LIN {X 0,Y 720.147,Z 331.518,A -85,B 0,C 180,E1 -1471.751,E2 -1471.751} C_VEL
LIN {X 0,Y 720.168,Z 331.521,A -85,B 0,C 180,E1 -1474.312,E2 -1474.312} C_VEL
LIN {X 0,Y 720.178,Z 331.516,A -85,B 0,C 180,E1 -1477.424,E2 -1477.424} C_VEL
LIN {X 0,Y 720.147,Z 331.52,A -85,B 0,C 180,E1 -1480.005,E2 -1480.005} C_VEL
LIN {X 0,Y 720.202,Z 331.519,A -85,B 0,C 180,E1 -1482.741,E2 -1482.741} C_VEL
LIN {X 0,Y 720.163,Z 331.518,A -85,B 0,C 180,E1 -1485.703,E2 -1485.703} C_VEL
LIN {X 0,Y 720.148,Z 331.521,A -85,B 0,C 180,E1 -1488.211,E2 -1488.211} C_VEL
LIN {X 0,Y 720.224,Z 331.522,A -85,B 0,C 180,E1 -1491.031,E2 -1491.031} C_VEL
LIN {X 0,Y 720.178,Z 331.658,A -85,B 0,C 180,E1 -1491.842,E2 -1491.842} C_VEL
LIN {X 0,Y 724.726,Z 343.938,A -85,B 0,C 180,E1 -1493.02,E2 -1493.02} C_VEL
LIN {X 0,Y 724.3,Z 377.38,A -85,B 0,C 180,E1 -1495.364,E2 -1495.364} C_VEL
LIN {X 0,Y 726.479,Z 386.984,A -85,B 0,C 180,E1 -1495.595,E2 -1495.595} C_VEL
LIN {X 0,Y 725.423,Z 646.459,A -85,B 0,C 180,E1 -1498.538,E2 -1498.538} C_VEL
LIN {X 0,Y 724.936,Z 767.067,A -85,B 0,C 180,E1 -1499.901,E2 -1499.901} C_VEL
LIN {X 0,Y 724.615,Z 792.768,A -85,B 0,C 180,E1 -1500.336,E2 -1500.336} C_VEL
LIN {X 0,Y 724.343,Z 814.337,A -85,B 0,C 180,E1 -1500.838,E2 -1500.838} C_VEL
LIN {X 0,Y 723.978,Z 838.571,A -85,B 0,C 180,E1 -1501.544,E2 -1501.544} C_VEL
LIN {X 0,Y 723.547,Z 860.481,A -85,B 0,C 180,E1 -1502.333,E2 -1502.333} C_VEL
LIN {X 0,Y 723.146,Z 883.179,A -85,B 0,C 180,E1 -1503.296,E2 -1503.296} C_VEL
LIN {X 0,Y 722.632,Z 904.752,A -85,B 0,C 180,E1 -1504.38,E2 -1504.38} C_VEL
LIN {X 0,Y 722.216,Z 925.848,A -85,B 0,C 180,E1 -1505.596,E2 -1505.596} C_VEL
LIN {X 0,Y 721.746,Z 945.564,A -85,B 0,C 180,E1 -1506.911,E2 -1506.911} C_VEL
LIN {X 0,Y 721.365,Z 964.778,A -85,B 0,C 180,E1 -1508.364,E2 -1508.364} C_VEL
LIN {X 0,Y 721.012,Z 981.391,A -85,B 0,C 180,E1 -1509.799,E2 -1509.799} C_VEL
LIN {X 0,Y 720.713,Z 998.517,A -85,B 0,C 180,E1 -1511.476,E2 -1511.476} C_VEL
LIN {X 0,Y 720.475,Z 1012.01,A -85,B 0,C 180,E1 -1512.982,E2 -1512.982} C_VEL
LIN {X 0,Y 720.287,Z 1026.218,A -85,B 0,C 180,E1 -1514.789,E2 -1514.789} C_VEL
LIN {X 0,Y 720.15,Z 1037.315,A -85,B 0,C 180,E1 -1516.429,E2 -1516.429} C_VEL
LIN {X 0,Y 720.044,Z 1047.962,A -85,B 0,C 180,E1 -1518.238,E2 -1518.238} C_VEL
LIN {X 0,Y 719.96,Z 1056.892,A -85,B 0,C 180,E1 -1520.083,E2 -1520.083} C_VEL
LIN {X 0,Y 719.941,Z 1063.423,A -85,B 0,C 180,E1 -1521.695,E2 -1521.695} C_VEL
LIN {X 0,Y 719.913,Z 1069.864,A -85,B 0,C 180,E1 -1523.701,E2 -1523.701} C_VEL
LIN {X 0,Y 719.916,Z 1073.813,A -85,B 0,C 180,E1 -1525.379,E2 -1525.379} C_VEL
LIN {X 0,Y 719.907,Z 1076.797,A -85,B 0,C 180,E1 -1527.214,E2 -1527.214} C_VEL
LIN {X 0,Y 719.9,Z 1078.284,A -85,B 0,C 180,E1 -1529.204,E2 -1529.204} C_VEL
LIN {X 0,Y 719.906,Z 1078.262,A -85,B 0,C 180,E1 -1530.875,E2 -1530.875} C_VEL
LIN {X 0,Y 719.913,Z 1076.572,A -85,B 0,C 180,E1 -1532.946,E2 -1532.946} C_VEL
LIN {X 0,Y 719.919,Z 1073.654,A -85,B 0,C 180,E1 -1534.7,E2 -1534.7} C_VEL
LIN {X 0,Y 719.908,Z 1069.015,A -85,B 0,C 180,E1 -1536.62,E2 -1536.62} C_VEL
LIN {X 0,Y 719.933,Z 1062.815,A -85,B 0,C 180,E1 -1538.466,E2 -1538.466} C_VEL
LIN {X 0,Y 719.974,Z 1056.182,A -85,B 0,C 180,E1 -1540.078,E2 -1540.078} C_VEL
LIN {X 0,Y 720.049,Z 1046.492,A -85,B 0,C 180,E1 -1542.023,E2 -1542.023} C_VEL
LIN {X 0,Y 720.154,Z 1036.797,A -85,B 0,C 180,E1 -1543.653,E2 -1543.653} C_VEL
LIN {X 0,Y 720.323,Z 1024.443,A -85,B 0,C 180,E1 -1545.457,E2 -1545.457} C_VEL
LIN {X 0,Y 720.483,Z 1011.22,A -85,B 0,C 180,E1 -1547.11,E2 -1547.11} C_VEL
LIN {X 0,Y 720.769,Z 996.177,A -85,B 0,C 180,E1 -1548.774,E2 -1548.774} C_VEL
LIN {X 0,Y 721.055,Z 979.533,A -85,B 0,C 180,E1 -1550.369,E2 -1550.369} C_VEL
LIN {X 0,Y 721.431,Z 961.605,A -85,B 0,C 180,E1 -1551.89,E2 -1551.89} C_VEL
LIN {X 0,Y 721.806,Z 943.237,A -85,B 0,C 180,E1 -1553.253,E2 -1553.253} C_VEL
LIN {X 0,Y 722.274,Z 921.436,A -85,B 0,C 180,E1 -1554.67,E2 -1554.67} C_VEL
LIN {X 0,Y 722.724,Z 901.528,A -85,B 0,C 180,E1 -1555.792,E2 -1555.792} C_VEL
LIN {X 0,Y 723.207,Z 878.257,A -85,B 0,C 180,E1 -1556.923,E2 -1556.923} C_VEL
LIN {X 0,Y 723.622,Z 857.111,A -85,B 0,C 180,E1 -1557.798,E2 -1557.798} C_VEL
LIN {X 0,Y 724.075,Z 832.965,A -85,B 0,C 180,E1 -1558.632,E2 -1558.632} C_VEL
LIN {X 0,Y 724.365,Z 811.104,A -85,B 0,C 180,E1 -1559.246,E2 -1559.246} C_VEL
LIN {X 0,Y 724.75,Z 786.45,A -85,B 0,C 180,E1 -1559.787,E2 -1559.787} C_VEL
LIN {X 0,Y 724.95,Z 763.827,A -85,B 0,C 180,E1 -1560.142,E2 -1560.142} C_VEL
LIN {X 0,Y 725.947,Z 508.76,A -85,B 0,C 180,E1 -1563.015,E2 -1563.015} C_VEL
LIN {X 0,Y 726.325,Z 385.42,A -85,B 0,C 180,E1 -1564.431,E2 -1564.431} C_VEL
LIN {X 0,Y 724.228,Z 376.685,A -85,B 0,C 180,E1 -1564.668,E2 -1564.668} C_VEL
LIN {X 0,Y 724.705,Z 343.756,A -85,B 0,C 180,E1 -1566.995,E2 -1566.995} C_VEL
LIN {X 0,Y 720.163,Z 331.523,A -85,B 0,C 180,E1 -1568.182,E2 -1568.182} C_VEL
LIN {X 0,Y 720.198,Z 331.524,A -85,B 0,C 180,E1 -1571.193,E2 -1571.193} C_VEL
LIN {X 0,Y 720.148,Z 331.521,A -85,B 0,C 180,E1 -1573.895,E2 -1573.895} C_VEL
LIN {X 0,Y 720.193,Z 331.517,A -85,B 0,C 180,E1 -1576.588,E2 -1576.588} C_VEL
LIN {X 0,Y 720.167,Z 331.519,A -85,B 0,C 180,E1 -1579.579,E2 -1579.579} C_VEL
LIN {X 0,Y 720.149,Z 331.518,A -85,B 0,C 180,E1 -1582.143,E2 -1582.143} C_VEL
LIN {X 0,Y 720.216,Z 331.516,A -85,B 0,C 180,E1 -1584.917,E2 -1584.917} C_VEL
LIN {X 0,Y 720.155,Z 331.519,A -85,B 0,C 180,E1 -1587.881,E2 -1587.881} C_VEL
LIN {X 0,Y 720.157,Z 331.517,A -85,B 0,C 180,E1 -1590.469,E2 -1590.469} C_VEL
LIN {X 0,Y 720.218,Z 331.517,A -85,B 0,C 180,E1 -1593.39,E2 -1593.39} C_VEL
LIN {X 0,Y 720.149,Z 331.515,A -85,B 0,C 180,E1 -1596.204,E2 -1596.204} C_VEL
LIN {X 0,Y 720.169,Z 331.516,A -85,B 0,C 180,E1 -1598.754,E2 -1598.754} C_VEL
LIN {X 0,Y 720.188,Z 331.521,A -85,B 0,C 180,E1 -1601.797,E2 -1601.797} C_VEL
LIN {X 0,Y 720.148,Z 331.517,A -85,B 0,C 180,E1 -1604.456,E2 -1604.456} C_VEL
LIN {X 0,Y 720.202,Z 331.513,A -85,B 0,C 180,E1 -1607.165,E2 -1607.165} C_VEL
LIN {X 0,Y 720.164,Z 331.515,A -85,B 0,C 180,E1 -1610.167,E2 -1610.167} C_VEL
LIN {X 0,Y 720.152,Z 331.517,A -85,B 0,C 180,E1 -1612.741,E2 -1612.741} C_VEL
LIN {X 0,Y 720.222,Z 331.515,A -85,B 0,C 180,E1 -1615.621,E2 -1615.621} C_VEL
LIN {X 0,Y 720.153,Z 331.519,A -85,B 0,C 180,E1 -1618.488,E2 -1618.488} C_VEL
LIN {X 0,Y 720.161,Z 331.511,A -85,B 0,C 180,E1 -1621.034,E2 -1621.034} C_VEL
LIN {X 0,Y 720.216,Z 331.521,A -85,B 0,C 180,E1 -1623.98,E2 -1623.98} C_VEL
LIN {X 0,Y 720.152,Z 331.517,A -85,B 0,C 180,E1 -1626.698,E2 -1626.698} C_VEL
LIN {X 0,Y 720.17,Z 331.516,A -85,B 0,C 180,E1 -1629.268,E2 -1629.268} C_VEL
LIN {X 0,Y 720.186,Z 331.521,A -85,B 0,C 180,E1 -1632.346,E2 -1632.346} C_VEL
LIN {X 0,Y 720.15,Z 331.516,A -85,B 0,C 180,E1 -1634.966,E2 -1634.966} C_VEL
LIN {X 0,Y 720.206,Z 331.518,A -85,B 0,C 180,E1 -1636.264,E2 -1636.264} C_VEL
LIN {X 0,Y 719.167,Z 331.649,A -85,B 0,C 180,E1 -1636.877,E2 -1636.877} C_VEL
LIN {X 0,Y 712.739,Z 332.448,A -85,B 0,C 180,E1 -1638.593,E2 -1638.593} C_VEL
LIN {X 0,Y 712.213,Z 332.507,A -85,B 0,C 180,E1 -1639.04,E2 -1639.04} C_VEL
LIN {X 0,Y 712.266,Z 332.499,A -85,B 0,C 180,E1 -1641.753,E2 -1641.753} C_VEL
LIN {X 0,Y 712.229,Z 332.504,A -85,B 0,C 180,E1 -1644.731,E2 -1644.731} C_VEL
LIN {X 0,Y 712.217,Z 332.506,A -85,B 0,C 180,E1 -1647.328,E2 -1647.328} C_VEL
LIN {X 0,Y 712.282,Z 332.501,A -85,B 0,C 180,E1 -1650.169,E2 -1650.169} C_VEL
LIN {X 0,Y 712.217,Z 332.505,A -85,B 0,C 180,E1 -1653.056,E2 -1653.056} C_VEL
LIN {X 0,Y 712.227,Z 332.505,A -85,B 0,C 180,E1 -1655.635,E2 -1655.635} C_VEL
LIN {X 0,Y 712.269,Z 332.51,A -85,B 0,C 180,E1 -1658.66,E2 -1658.66} C_VEL
LIN {X 0,Y 712.215,Z 332.509,A -85,B 0,C 180,E1 -1661.395,E2 -1661.395} C_VEL
LIN {X 0,Y 712.27,Z 332.495,A -85,B 0,C 180,E1 -1664.164,E2 -1664.164} C_VEL
LIN {X 0,Y 712.23,Z 332.509,A -85,B 0,C 180,E1 -1667.124,E2 -1667.124} C_VEL
LIN {X 0,Y 712.222,Z 332.508,A -85,B 0,C 180,E1 -1669.775,E2 -1669.775} C_VEL
LIN {X 0,Y 712.284,Z 332.51,A -85,B 0,C 180,E1 -1672.745,E2 -1672.745} C_VEL
LIN {X 0,Y 712.233,Z 332.633,A -85,B 0,C 180,E1 -1675.569,E2 -1675.569} C_VEL
LIN {X 0,Y 716.874,Z 346.258,A -85,B 0,C 180,E1 -1676.903,E2 -1676.903} C_VEL
LIN {X 0,Y 717.012,Z 348.148,A -85,B 0,C 180,E1 -1677.015,E2 -1677.015} C_VEL
LIN {X 0,Y 719.82,Z 359.326,A -85,B 0,C 180,E1 -1677.304,E2 -1677.304} C_VEL
LIN {X 0,Y 718.694,Z 595.051,A -85,B 0,C 180,E1 -1680.007,E2 -1680.007} C_VEL
LIN {X 0,Y 718.005,Z 736.964,A -85,B 0,C 180,E1 -1681.623,E2 -1681.623} C_VEL
LIN {X 0,Y 717.641,Z 762.526,A -85,B 0,C 180,E1 -1682.058,E2 -1682.058} C_VEL
LIN {X 0,Y 717.294,Z 784.203,A -85,B 0,C 180,E1 -1682.564,E2 -1682.564} C_VEL
LIN {X 0,Y 716.87,Z 808.198,A -85,B 0,C 180,E1 -1683.268,E2 -1683.268} C_VEL
LIN {X 0,Y 716.361,Z 829.733,A -85,B 0,C 180,E1 -1684.046,E2 -1684.046} C_VEL
LIN {X 0,Y 715.863,Z 852.405,A -85,B 0,C 180,E1 -1685.011,E2 -1685.011} C_VEL
LIN {X 0,Y 715.255,Z 874.42,A -85,B 0,C 180,E1 -1686.123,E2 -1686.123} C_VEL
LIN {X 0,Y 714.733,Z 895.263,A -85,B 0,C 180,E1 -1687.33,E2 -1687.33} C_VEL
LIN {X 0,Y 714.192,Z 914.96,A -85,B 0,C 180,E1 -1688.653,E2 -1688.653} C_VEL
LIN {X 0,Y 713.716,Z 933.972,A -85,B 0,C 180,E1 -1690.097,E2 -1690.097} C_VEL
LIN {X 0,Y 713.27,Z 951.38,A -85,B 0,C 180,E1 -1691.614,E2 -1691.614} C_VEL
LIN {X 0,Y 712.899,Z 968.676,A -85,B 0,C 180,E1 -1693.327,E2 -1693.327} C_VEL
LIN {X 0,Y 712.588,Z 983.029,A -85,B 0,C 180,E1 -1694.954,E2 -1694.954} C_VEL
LIN {X 0,Y 712.339,Z 997.581,A -85,B 0,C 180,E1 -1696.856,E2 -1696.856} C_VEL
LIN {X 0,Y 712.188,Z 1008.453,A -85,B 0,C 180,E1 -1698.5,E2 -1698.5} C_VEL
LIN {X 0,Y 712.068,Z 1019.527,A -85,B 0,C 180,E1 -1700.462,E2 -1700.462} C_VEL
LIN {X 0,Y 711.974,Z 1027.563,A -85,B 0,C 180,E1 -1702.171,E2 -1702.171} C_VEL
LIN {X 0,Y 711.944,Z 1034.871,A -85,B 0,C 180,E1 -1704.035,E2 -1704.035} C_VEL
LIN {X 0,Y 711.926,Z 1040.624,A -85,B 0,C 180,E1 -1705.973,E2 -1705.973} C_VEL
LIN {X 0,Y 711.916,Z 1044.548,A -85,B 0,C 180,E1 -1707.746,E2 -1707.746} C_VEL
LIN {X 0,Y 711.919,Z 1047.404,A -85,B 0,C 180,E1 -1709.839,E2 -1709.839} C_VEL
LIN {X 0,Y 711.89,Z 1048.364,A -85,B 0,C 180,E1 -1711.529,E2 -1711.529} C_VEL
LIN {X 0,Y 711.901,Z 1048.059,A -85,B 0,C 180,E1 -1713.462,E2 -1713.462} C_VEL
LIN {X 0,Y 711.906,Z 1046.161,A -85,B 0,C 180,E1 -1715.319,E2 -1715.319} C_VEL
LIN {X 0,Y 711.921,Z 1043.062,A -85,B 0,C 180,E1 -1717.1,E2 -1717.1} C_VEL
LIN {X 0,Y 711.935,Z 1037.783,A -85,B 0,C 180,E1 -1719.132,E2 -1719.132} C_VEL
LIN {X 0,Y 711.938,Z 1032.221,A -85,B 0,C 180,E1 -1720.766,E2 -1720.766} C_VEL
LIN {X 0,Y 712.017,Z 1024.357,A -85,B 0,C 180,E1 -1722.655,E2 -1722.655} C_VEL
LIN {X 0,Y 712.112,Z 1014.976,A -85,B 0,C 180,E1 -1724.474,E2 -1724.474} C_VEL
LIN {X 0,Y 712.25,Z 1004.476,A -85,B 0,C 180,E1 -1726.222,E2 -1726.222} C_VEL
LIN {X 0,Y 712.441,Z 991.458,A -85,B 0,C 180,E1 -1728.069,E2 -1728.069} C_VEL
LIN {X 0,Y 712.708,Z 978.141,A -85,B 0,C 180,E1 -1729.715,E2 -1729.715} C_VEL
LIN {X 0,Y 713.004,Z 962.68,A -85,B 0,C 180,E1 -1731.384,E2 -1731.384} C_VEL
LIN {X 0,Y 713.401,Z 946.869,A -85,B 0,C 180,E1 -1732.889,E2 -1732.889} C_VEL
LIN {X 0,Y 713.83,Z 928.46,A -85,B 0,C 180,E1 -1734.427,E2 -1734.427} C_VEL
LIN {X 0,Y 714.333,Z 910.388,A -85,B 0,C 180,E1 -1735.761,E2 -1735.761} C_VEL
LIN {X 0,Y 714.844,Z 889.874,A -85,B 0,C 180,E1 -1737.084,E2 -1737.084} C_VEL
LIN {X 0,Y 715.391,Z 870.255,A -85,B 0,C 180,E1 -1738.191,E2 -1738.191} C_VEL
LIN {X 0,Y 715.937,Z 847.27,A -85,B 0,C 180,E1 -1739.309,E2 -1739.309} C_VEL
LIN {X 0,Y 716.445,Z 826.736,A -85,B 0,C 180,E1 -1740.161,E2 -1740.161} C_VEL
LIN {X 0,Y 716.974,Z 802.732,A -85,B 0,C 180,E1 -1740.994,E2 -1740.994} C_VEL
LIN {X 0,Y 717.328,Z 781.027,A -85,B 0,C 180,E1 -1741.608,E2 -1741.608} C_VEL
LIN {X 0,Y 717.788,Z 756.2,A -85,B 0,C 180,E1 -1742.155,E2 -1742.155} C_VEL
LIN {X 0,Y 718.022,Z 733.611,A -85,B 0,C 180,E1 -1742.511,E2 -1742.511} C_VEL
LIN {X 0,Y 719.275,Z 474.158,A -85,B 0,C 180,E1 -1745.46,E2 -1745.46} C_VEL
LIN {X 0,Y 719.66,Z 357.915,A -85,B 0,C 180,E1 -1746.811,E2 -1746.811} C_VEL
LIN {X 0,Y 716.859,Z 347.284,A -85,B 0,C 180,E1 -1747.109,E2 -1747.109} C_VEL
LIN {X 0,Y 716.355,Z 344.494,A -85,B 0,C 180,E1 -1747.353,E2 -1747.353} C_VEL
LIN {X 0,Y 712.215,Z 332.516,A -85,B 0,C 180,E1 -1748.56,E2 -1748.56} C_VEL
LIN {X 0,Y 712.284,Z 332.508,A -85,B 0,C 180,E1 -1751.442,E2 -1751.442} C_VEL
LIN {X 0,Y 712.216,Z 332.507,A -85,B 0,C 180,E1 -1754.359,E2 -1754.359} C_VEL
LIN {X 0,Y 712.233,Z 332.509,A -85,B 0,C 180,E1 -1757.006,E2 -1757.006} C_VEL
LIN {X 0,Y 712.245,Z 332.502,A -85,B 0,C 180,E1 -1760.091,E2 -1760.091} C_VEL
LIN {X 0,Y 712.213,Z 332.508,A -85,B 0,C 180,E1 -1762.752,E2 -1762.752} C_VEL
LIN {X 0,Y 712.278,Z 332.503,A -85,B 0,C 180,E1 -1765.547,E2 -1765.547} C_VEL
LIN {X 0,Y 712.219,Z 332.503,A -85,B 0,C 180,E1 -1768.516,E2 -1768.516} C_VEL
LIN {X 0,Y 712.224,Z 332.509,A -85,B 0,C 180,E1 -1771.122,E2 -1771.122} C_VEL
LIN {X 0,Y 712.272,Z 332.501,A -85,B 0,C 180,E1 -1774.114,E2 -1774.114} C_VEL
LIN {X 0,Y 712.213,Z 332.507,A -85,B 0,C 180,E1 -1776.863,E2 -1776.863} C_VEL
LIN {X 0,Y 712.249,Z 332.508,A -85,B 0,C 180,E1 -1779.54,E2 -1779.54} C_VEL
LIN {X 0,Y 712.23,Z 332.503,A -85,B 0,C 180,E1 -1782.601,E2 -1782.601} C_VEL
LIN {X 0,Y 712.213,Z 332.508,A -85,B 0,C 180,E1 -1785.196,E2 -1785.196} C_VEL
LIN {X 0,Y 712.283,Z 332.507,A -85,B 0,C 180,E1 -1788.079,E2 -1788.079} C_VEL
LIN {X 0,Y 712.216,Z 332.505,A -85,B 0,C 180,E1 -1790.953,E2 -1790.953} C_VEL
LIN {X 0,Y 712.225,Z 332.509,A -85,B 0,C 180,E1 -1793.551,E2 -1793.551} C_VEL
LIN {X 0,Y 712.266,Z 332.504,A -85,B 0,C 180,E1 -1796.539,E2 -1796.539} C_VEL
LIN {X 0,Y 712.21,Z 332.504,A -85,B 0,C 180,E1 -1799.276,E2 -1799.276} C_VEL
LIN {X 0,Y 712.249,Z 332.511,A -85,B 0,C 180,E1 -1801.931,E2 -1801.931} C_VEL
LIN {X 0,Y 712.228,Z 332.505,A -85,B 0,C 180,E1 -1804.993,E2 -1804.993} C_VEL
LIN {X 0,Y 712.211,Z 332.504,A -85,B 0,C 180,E1 -1807.583,E2 -1807.583} C_VEL
LIN {X 0,Y 712.283,Z 332.504,A -85,B 0,C 180,E1 -1810.433,E2 -1810.433} C_VEL
LIN {X 0,Y 712.216,Z 332.506,A -85,B 0,C 180,E1 -1813.311,E2 -1813.311} C_VEL
LIN {X 0,Y 712.221,Z 332.505,A -85,B 0,C 180,E1 -1815.914,E2 -1815.914} C_VEL
LIN {X 0,Y 712.263,Z 332.499,A -85,B 0,C 180,E1 -1818.922,E2 -1818.922} C_VEL
LIN {X 0,Y 712.209,Z 332.507,A -85,B 0,C 180,E1 -1821.668,E2 -1821.668} C_VEL
LIN {X 0,Y 712.252,Z 332.507,A -85,B 0,C 180,E1 -1824.343,E2 -1824.343} C_VEL
LIN {X 0,Y 712.231,Z 332.503,A -85,B 0,C 180,E1 -1827.327,E2 -1827.327} C_VEL
LIN {X 0,Y 712.209,Z 332.508,A -85,B 0,C 180,E1 -1829.894,E2 -1829.894} C_VEL
LIN {X 0,Y 712.28,Z 332.51,A -85,B 0,C 180,E1 -1832.715,E2 -1832.715} C_VEL
LIN {X 0,Y 712.218,Z 332.507,A -85,B 0,C 180,E1 -1835.635,E2 -1835.635} C_VEL
LIN {X 0,Y 712.214,Z 332.509,A -85,B 0,C 180,E1 -1838.169,E2 -1838.169} C_VEL
LIN {X 0,Y 712.283,Z 332.506,A -85,B 0,C 180,E1 -1841.077,E2 -1841.077} C_VEL
LIN {X 0,Y 712.21,Z 332.508,A -85,B 0,C 180,E1 -1843.928,E2 -1843.928} C_VEL
LIN {X 0,Y 712.231,Z 332.512,A -85,B 0,C 180,E1 -1846.537,E2 -1846.537} C_VEL
LIN {X 0,Y 712.234,Z 332.511,A -85,B 0,C 180,E1 -1849.67,E2 -1849.67} C_VEL
LIN {X 0,Y 712.304,Z 332.749,A -85,B 0,C 180,E1 -1851.434,E2 -1851.434} C_VEL
LIN {X 0,Y 717.694,Z 347.211,A -85,B 0,C 180,E1 -1852.836,E2 -1852.836} C_VEL
LIN {X 0,Y 717.276,Z 377.475,A -85,B 0,C 180,E1 -1854.976,E2 -1854.976} C_VEL
LIN {X 0,Y 719.862,Z 388.77,A -85,B 0,C 180,E1 -1855.255,E2 -1855.255} C_VEL
LIN {X 0,Y 718.585,Z 648.445,A -85,B 0,C 180,E1 -1858.226,E2 -1858.226} C_VEL
LIN {X 0,Y 718.004,Z 767.174,A -85,B 0,C 180,E1 -1859.581,E2 -1859.581} C_VEL
LIN {X 0,Y 717.629,Z 792.895,A -85,B 0,C 180,E1 -1860.021,E2 -1860.021} C_VEL
LIN {X 0,Y 717.291,Z 814.459,A -85,B 0,C 180,E1 -1860.526,E2 -1860.526} C_VEL
LIN {X 0,Y 716.861,Z 838.568,A -85,B 0,C 180,E1 -1861.235,E2 -1861.235} C_VEL
LIN {X 0,Y 716.339,Z 860.486,A -85,B 0,C 180,E1 -1862.031,E2 -1862.031} C_VEL
LIN {X 0,Y 715.831,Z 883.582,A -85,B 0,C 180,E1 -1863.022,E2 -1863.022} C_VEL
LIN {X 0,Y 715.246,Z 904.756,A -85,B 0,C 180,E1 -1864.096,E2 -1864.096} C_VEL
LIN {X 0,Y 714.719,Z 925.755,A -85,B 0,C 180,E1 -1865.317,E2 -1865.317} C_VEL
LIN {X 0,Y 714.177,Z 945.152,A -85,B 0,C 180,E1 -1866.622,E2 -1866.622} C_VEL
LIN {X 0,Y 713.724,Z 963.809,A -85,B 0,C 180,E1 -1868.038,E2 -1868.038} C_VEL
LIN {X 0,Y 713.296,Z 980.462,A -85,B 0,C 180,E1 -1869.485,E2 -1869.485} C_VEL
LIN {X 0,Y 712.938,Z 996.965,A -85,B 0,C 180,E1 -1871.096,E2 -1871.096} C_VEL
LIN {X 0,Y 712.623,Z 1011.222,A -85,B 0,C 180,E1 -1872.695,E2 -1872.695} C_VEL
LIN {X 0,Y 712.408,Z 1025.06,A -85,B 0,C 180,E1 -1874.45,E2 -1874.45} C_VEL
LIN {X 0,Y 712.209,Z 1036.797,A -85,B 0,C 180,E1 -1876.192,E2 -1876.192} C_VEL
LIN {X 0,Y 712.082,Z 1046.948,A -85,B 0,C 180,E1 -1877.923,E2 -1877.923} C_VEL
LIN {X 0,Y 711.99,Z 1056.524,A -85,B 0,C 180,E1 -1879.886,E2 -1879.886} C_VEL
LIN {X 0,Y 711.94,Z 1063.12,A -85,B 0,C 180,E1 -1881.52,E2 -1881.52} C_VEL
LIN {X 0,Y 711.909,Z 1069.451,A -85,B 0,C 180,E1 -1883.468,E2 -1883.468} C_VEL
LIN {X 0,Y 711.918,Z 1073.814,A -85,B 0,C 180,E1 -1885.327,E2 -1885.327} C_VEL
LIN {X 0,Y 711.908,Z 1076.797,A -85,B 0,C 180,E1 -1887.182,E2 -1887.182} C_VEL
LIN {X 0,Y 711.901,Z 1078.284,A -85,B 0,C 180,E1 -1889.195,E2 -1889.195} C_VEL
LIN {X 0,Y 711.906,Z 1078.262,A -85,B 0,C 180,E1 -1890.885,E2 -1890.885} C_VEL
LIN {X 0,Y 711.914,Z 1076.572,A -85,B 0,C 180,E1 -1892.979,E2 -1892.979} C_VEL
LIN {X 0,Y 711.919,Z 1073.655,A -85,B 0,C 180,E1 -1894.753,E2 -1894.753} C_VEL
LIN {X 0,Y 711.914,Z 1069.015,A -85,B 0,C 180,E1 -1896.694,E2 -1896.694} C_VEL
LIN {X 0,Y 711.938,Z 1062.815,A -85,B 0,C 180,E1 -1898.562,E2 -1898.562} C_VEL
LIN {X 0,Y 712.001,Z 1056.182,A -85,B 0,C 180,E1 -1900.192,E2 -1900.192} C_VEL
LIN {X 0,Y 712.095,Z 1046.032,A -85,B 0,C 180,E1 -1902.241,E2 -1902.241} C_VEL
LIN {X 0,Y 712.214,Z 1036.279,A -85,B 0,C 180,E1 -1903.891,E2 -1903.891} C_VEL
LIN {X 0,Y 712.423,Z 1023.806,A -85,B 0,C 180,E1 -1905.716,E2 -1905.716} C_VEL
LIN {X 0,Y 712.64,Z 1010.515,A -85,B 0,C 180,E1 -1907.389,E2 -1907.389} C_VEL
LIN {X 0,Y 712.961,Z 995.334,A -85,B 0,C 180,E1 -1909.073,E2 -1909.073} C_VEL
LIN {X 0,Y 713.319,Z 979.534,A -85,B 0,C 180,E1 -1910.6,E2 -1910.6} C_VEL
LIN {X 0,Y 713.767,Z 961.606,A -85,B 0,C 180,E1 -1912.138,E2 -1912.138} C_VEL
LIN {X 0,Y 714.239,Z 943.237,A -85,B 0,C 180,E1 -1913.515,E2 -1913.515} C_VEL
LIN {X 0,Y 714.782,Z 922.166,A -85,B 0,C 180,E1 -1914.902,E2 -1914.902} C_VEL
LIN {X 0,Y 715.321,Z 902.334,A -85,B 0,C 180,E1 -1916.035,E2 -1916.035} C_VEL
LIN {X 0,Y 715.904,Z 879.254,A -85,B 0,C 180,E1 -1917.175,E2 -1917.175} C_VEL
LIN {X 0,Y 716.401,Z 858.239,A -85,B 0,C 180,E1 -1918.057,E2 -1918.057} C_VEL
LIN {X 0,Y 716.951,Z 834.438,A -85,B 0,C 180,E1 -1918.897,E2 -1918.897} C_VEL
LIN {X 0,Y 717.314,Z 811.86,A -85,B 0,C 180,E1 -1919.542,E2 -1919.542} C_VEL
LIN {X 0,Y 717.775,Z 787.537,A -85,B 0,C 180,E1 -1920.087,E2 -1920.087} C_VEL
LIN {X 0,Y 718.02,Z 764.114,A -85,B 0,C 180,E1 -1920.459,E2 -1920.459} C_VEL
LIN {X 0,Y 719.22,Z 511.246,A -85,B 0,C 180,E1 -1923.334,E2 -1923.334} C_VEL
LIN {X 0,Y 719.678,Z 387.124,A -85,B 0,C 180,E1 -1924.775,E2 -1924.775} C_VEL
LIN {X 0,Y 717.183,Z 376.685,A -85,B 0,C 180,E1 -1925.058,E2 -1925.058} C_VEL
LIN {X 0,Y 717.695,Z 347.209,A -85,B 0,C 180,E1 -1927.164,E2 -1927.164} C_VEL
LIN {X 0,Y 712.276,Z 332.509,A -85,B 0,C 180,E1 -1928.608,E2 -1928.608} C_VEL
LIN {X 0,Y 712.219,Z 332.513,A -85,B 0,C 180,E1 -1931.558,E2 -1931.558} C_VEL
LIN {X 0,Y 712.214,Z 332.51,A -85,B 0,C 180,E1 -1934.134,E2 -1934.134} C_VEL
LIN {X 0,Y 712.281,Z 332.51,A -85,B 0,C 180,E1 -1937.001,E2 -1937.001} C_VEL
LIN {X 0,Y 712.213,Z 332.507,A -85,B 0,C 180,E1 -1939.794,E2 -1939.794} C_VEL
LIN {X 0,Y 712.219,Z 332.506,A -85,B 0,C 180,E1 -1942.36,E2 -1942.36} C_VEL
LIN {X 0,Y 712.271,Z 332.507,A -85,B 0,C 180,E1 -1945.351,E2 -1945.351} C_VEL
LIN {X 0,Y 712.209,Z 332.507,A -85,B 0,C 180,E1 -1948.043,E2 -1948.043} C_VEL
LIN {X 0,Y 712.234,Z 332.505,A -85,B 0,C 180,E1 -1950.669,E2 -1950.669} C_VEL
LIN {X 0,Y 712.236,Z 332.51,A -85,B 0,C 180,E1 -1953.776,E2 -1953.776} C_VEL
LIN {X 0,Y 712.211,Z 332.503,A -85,B 0,C 180,E1 -1956.414,E2 -1956.414} C_VEL
LIN {X 0,Y 712.282,Z 332.504,A -85,B 0,C 180,E1 -1959.215,E2 -1959.215} C_VEL
LIN {X 0,Y 712.218,Z 332.508,A -85,B 0,C 180,E1 -1962.148,E2 -1962.148} C_VEL
LIN {X 0,Y 712.218,Z 332.504,A -85,B 0,C 180,E1 -1964.696,E2 -1964.696} C_VEL
LIN {X 0,Y 712.282,Z 332.508,A -85,B 0,C 180,E1 -1967.597,E2 -1967.597} C_VEL
LIN {X 0,Y 712.212,Z 332.503,A -85,B 0,C 180,E1 -1970.383,E2 -1970.383} C_VEL
LIN {X 0,Y 712.231,Z 332.505,A -85,B 0,C 180,E1 -1973,E2 -1973} C_VEL
LIN {X 0,Y 712.238,Z 332.508,A -85,B 0,C 180,E1 -1976.136,E2 -1976.136} C_VEL
LIN {X 0,Y 712.214,Z 332.506,A -85,B 0,C 180,E1 -1978.793,E2 -1978.793} C_VEL
LIN {X 0,Y 712.283,Z 332.498,A -85,B 0,C 180,E1 -1981.609,E2 -1981.609} C_VEL
LIN {X 0,Y 712.219,Z 332.506,A -85,B 0,C 180,E1 -1984.509,E2 -1984.509} C_VEL
LIN {X 0,Y 712.22,Z 332.503,A -85,B 0,C 180,E1 -1987.097,E2 -1987.097} C_VEL
LIN {X 0,Y 712.28,Z 332.507,A -85,B 0,C 180,E1 -1990.025,E2 -1990.025} C_VEL
LIN {X 0,Y 712.213,Z 332.507,A -85,B 0,C 180,E1 -1992.816,E2 -1992.816} C_VEL
LIN {X 0,Y 712.233,Z 332.503,A -85,B 0,C 180,E1 -1995.387,E2 -1995.387} C_VEL
LIN {X 0,Y 712.242,Z 332.51,A -85,B 0,C 180,E1 -1998.498,E2 -1998.498} C_VEL
LIN {X 0,Y 712.213,Z 332.507,A -85,B 0,C 180,E1 -1999.04,E2 -1999.04} C_VEL
LIN {X 0,Y 711.228,Z 332.632,A -85,B 0,C 180,E1 -1999.659,E2 -1999.659} C_VEL
LIN {X 0,Y 704.842,Z 333.422,A -85,B 0,C 180,E1 -2001.395,E2 -2001.395} C_VEL
LIN {X 0,Y 704.336,Z 333.488,A -85,B 0,C 180,E1 -2001.847,E2 -2001.847} C_VEL
LIN {X 0,Y 704.281,Z 333.492,A -85,B 0,C 180,E1 -2004.85,E2 -2004.85} C_VEL
LIN {X 0,Y 704.286,Z 333.495,A -85,B 0,C 180,E1 -2007.478,E2 -2007.478} C_VEL
LIN {X 0,Y 704.333,Z 333.498,A -85,B 0,C 180,E1 -2010.491,E2 -2010.491} C_VEL
LIN {X 0,Y 704.275,Z 333.492,A -85,B 0,C 180,E1 -2013.256,E2 -2013.256} C_VEL
LIN {X 0,Y 704.328,Z 333.493,A -85,B 0,C 180,E1 -2015.996,E2 -2015.996} C_VEL
LIN {X 0,Y 704.286,Z 333.497,A -85,B 0,C 180,E1 -2019.051,E2 -2019.051} C_VEL
LIN {X 0,Y 704.284,Z 333.497,A -85,B 0,C 180,E1 -2021.688,E2 -2021.688} C_VEL
LIN {X 0,Y 704.338,Z 333.483,A -85,B 0,C 180,E1 -2024.665,E2 -2024.665} C_VEL
LIN {X 0,Y 704.278,Z 333.495,A -85,B 0,C 180,E1 -2027.484,E2 -2027.484} C_VEL
LIN {X 0,Y 704.322,Z 333.495,A -85,B 0,C 180,E1 -2030.189,E2 -2030.189} C_VEL
LIN {X 0,Y 704.296,Z 333.504,A -85,B 0,C 180,E1 -2033.199,E2 -2033.199} C_VEL
LIN {X 0,Y 704.318,Z 333.634,A -85,B 0,C 180,E1 -2035.172,E2 -2035.172} C_VEL
LIN {X 0,Y 709.413,Z 347.994,A -85,B 0,C 180,E1 -2036.582,E2 -2036.582} C_VEL
LIN {X 0,Y 710.976,Z 352.032,A -85,B 0,C 180,E1 -2036.72,E2 -2036.72} C_VEL
LIN {X 0,Y 713.228,Z 361.214,A -85,B 0,C 180,E1 -2036.959,E2 -2036.959} C_VEL
LIN {X 0,Y 711.899,Z 596.712,A -85,B 0,C 180,E1 -2039.683,E2 -2039.683} C_VEL
LIN {X 0,Y 711.095,Z 737.104,A -85,B 0,C 180,E1 -2041.298,E2 -2041.298} C_VEL
LIN {X 0,Y 710.683,Z 762.688,A -85,B 0,C 180,E1 -2041.738,E2 -2041.738} C_VEL
LIN {X 0,Y 710.264,Z 784.444,A -85,B 0,C 180,E1 -2042.25,E2 -2042.25} C_VEL
LIN {X 0,Y 709.748,Z 808.927,A -85,B 0,C 180,E1 -2042.978,E2 -2042.978} C_VEL
LIN {X 0,Y 709.162,Z 830.486,A -85,B 0,C 180,E1 -2043.767,E2 -2043.767} C_VEL
LIN {X 0,Y 708.547,Z 853.569,A -85,B 0,C 180,E1 -2044.766,E2 -2044.766} C_VEL
LIN {X 0,Y 707.876,Z 874.78,A -85,B 0,C 180,E1 -2045.852,E2 -2045.852} C_VEL
LIN {X 0,Y 707.217,Z 896.311,A -85,B 0,C 180,E1 -2047.12,E2 -2047.12} C_VEL
LIN {X 0,Y 706.618,Z 915.313,A -85,B 0,C 180,E1 -2048.413,E2 -2048.413} C_VEL
LIN {X 0,Y 706.049,Z 934.283,A -85,B 0,C 180,E1 -2049.873,E2 -2049.873} C_VEL
LIN {X 0,Y 705.564,Z 950.732,A -85,B 0,C 180,E1 -2051.32,E2 -2051.32} C_VEL
LIN {X 0,Y 705.13,Z 967.025,A -85,B 0,C 180,E1 -2052.931,E2 -2052.931} C_VEL
LIN {X 0,Y 704.75,Z 981.839,A -85,B 0,C 180,E1 -2054.614,E2 -2054.614} C_VEL
LIN {X 0,Y 704.487,Z 995.453,A -85,B 0,C 180,E1 -2056.373,E2 -2056.373} C_VEL
LIN {X 0,Y 704.269,Z 1007.058,A -85,B 0,C 180,E1 -2058.12,E2 -2058.12} C_VEL
LIN {X 0,Y 704.119,Z 1017.561,A -85,B 0,C 180,E1 -2059.941,E2 -2059.941} C_VEL
LIN {X 0,Y 704.013,Z 1026.732,A -85,B 0,C 180,E1 -2061.864,E2 -2061.864} C_VEL
LIN {X 0,Y 703.947,Z 1033.449,A -85,B 0,C 180,E1 -2063.557,E2 -2063.557} C_VEL
LIN {X 0,Y 703.921,Z 1040.067,A -85,B 0,C 180,E1 -2065.682,E2 -2065.682} C_VEL
LIN {X 0,Y 703.915,Z 1043.96,A -85,B 0,C 180,E1 -2067.395,E2 -2067.395} C_VEL
LIN {X 0,Y 703.899,Z 1046.897,A -85,B 0,C 180,E1 -2069.267,E2 -2069.267} C_VEL
LIN {X 0,Y 703.9,Z 1048.281,A -85,B 0,C 180,E1 -2071.221,E2 -2071.221} C_VEL
LIN {X 0,Y 703.906,Z 1048.264,A -85,B 0,C 180,E1 -2072.931,E2 -2072.931} C_VEL
LIN {X 0,Y 703.911,Z 1046.58,A -85,B 0,C 180,E1 -2075.053,E2 -2075.053} C_VEL
LIN {X 0,Y 703.91,Z 1043.716,A -85,B 0,C 180,E1 -2076.821,E2 -2076.821} C_VEL
LIN {X 0,Y 703.925,Z 1039.223,A -85,B 0,C 180,E1 -2078.742,E2 -2078.742} C_VEL
LIN {X 0,Y 703.944,Z 1033.051,A -85,B 0,C 180,E1 -2080.641,E2 -2080.641} C_VEL
LIN {X 0,Y 704.021,Z 1026.412,A -85,B 0,C 180,E1 -2082.3,E2 -2082.3} C_VEL
LIN {X 0,Y 704.132,Z 1016.7,A -85,B 0,C 180,E1 -2084.305,E2 -2084.305} C_VEL
LIN {X 0,Y 704.274,Z 1006.757,A -85,B 0,C 180,E1 -2086.018,E2 -2086.018} C_VEL
LIN {X 0,Y 704.507,Z 994.482,A -85,B 0,C 180,E1 -2087.852,E2 -2087.852} C_VEL
LIN {X 0,Y 704.771,Z 981.118,A -85,B 0,C 180,E1 -2089.562,E2 -2089.562} C_VEL
LIN {X 0,Y 705.153,Z 965.849,A -85,B 0,C 180,E1 -2091.285,E2 -2091.285} C_VEL
LIN {X 0,Y 705.59,Z 949.887,A -85,B 0,C 180,E1 -2092.848,E2 -2092.848} C_VEL
LIN {X 0,Y 706.101,Z 932.311,A -85,B 0,C 180,E1 -2094.38,E2 -2094.38} C_VEL
LIN {X 0,Y 706.671,Z 913.726,A -85,B 0,C 180,E1 -2095.791,E2 -2095.791} C_VEL
LIN {X 0,Y 707.3,Z 893.136,A -85,B 0,C 180,E1 -2097.169,E2 -2097.169} C_VEL
LIN {X 0,Y 707.937,Z 873.068,A -85,B 0,C 180,E1 -2098.331,E2 -2098.331} C_VEL
LIN {X 0,Y 708.616,Z 850.437,A -85,B 0,C 180,E1 -2099.469,E2 -2099.469} C_VEL
LIN {X 0,Y 709.191,Z 829.539,A -85,B 0,C 180,E1 -2100.36,E2 -2100.36} C_VEL
LIN {X 0,Y 709.837,Z 806.353,A -85,B 0,C 180,E1 -2101.2,E2 -2101.2} C_VEL
LIN {X 0,Y 710.287,Z 782.585,A -85,B 0,C 180,E1 -2101.889,E2 -2101.889} C_VEL
LIN {X 0,Y 710.813,Z 758.633,A -85,B 0,C 180,E1 -2102.437,E2 -2102.437} C_VEL
LIN {X 0,Y 711.111,Z 734.559,A -85,B 0,C 180,E1 -2102.826,E2 -2102.826} C_VEL
LIN {X 0,Y 712.578,Z 476.432,A -85,B 0,C 180,E1 -2105.789,E2 -2105.789} C_VEL
LIN {X 0,Y 713.043,Z 359.592,A -85,B 0,C 180,E1 -2107.161,E2 -2107.161} C_VEL
LIN {X 0,Y 709.987,Z 349.207,A -85,B 0,C 180,E1 -2107.461,E2 -2107.461} C_VEL
LIN {X 0,Y 709.008,Z 347.055,A -85,B 0,C 180,E1 -2107.573,E2 -2107.573} C_VEL
LIN {X 0,Y 704.303,Z 333.503,A -85,B 0,C 180,E1 -2108.943,E2 -2108.943} C_VEL
LIN {X 0,Y 704.295,Z 333.498,A -85,B 0,C 180,E1 -2112.075,E2 -2112.075} C_VEL
LIN {X 0,Y 704.277,Z 333.497,A -85,B 0,C 180,E1 -2114.66,E2 -2114.66} C_VEL
LIN {X 0,Y 704.344,Z 333.496,A -85,B 0,C 180,E1 -2117.489,E2 -2117.489} C_VEL
LIN {X 0,Y 704.281,Z 333.492,A -85,B 0,C 180,E1 -2120.397,E2 -2120.397} C_VEL
LIN {X 0,Y 704.286,Z 333.498,A -85,B 0,C 180,E1 -2122.989,E2 -2122.989} C_VEL
LIN {X 0,Y 704.331,Z 333.493,A -85,B 0,C 180,E1 -2126.003,E2 -2126.003} C_VEL
LIN {X 0,Y 704.274,Z 333.493,A -85,B 0,C 180,E1 -2128.788,E2 -2128.788} C_VEL
LIN {X 0,Y 704.324,Z 333.498,A -85,B 0,C 180,E1 -2131.51,E2 -2131.51} C_VEL
LIN {X 0,Y 704.284,Z 333.492,A -85,B 0,C 180,E1 -2134.548,E2 -2134.548} C_VEL
LIN {X 0,Y 704.279,Z 333.498,A -85,B 0,C 180,E1 -2137.133,E2 -2137.133} C_VEL
LIN {X 0,Y 704.345,Z 333.493,A -85,B 0,C 180,E1 -2140.08,E2 -2140.08} C_VEL
LIN {X 0,Y 704.274,Z 333.494,A -85,B 0,C 180,E1 -2142.909,E2 -2142.909} C_VEL
LIN {X 0,Y 704.296,Z 333.498,A -85,B 0,C 180,E1 -2145.53,E2 -2145.53} C_VEL
LIN {X 0,Y 704.301,Z 333.493,A -85,B 0,C 180,E1 -2148.619,E2 -2148.619} C_VEL
LIN {X 0,Y 704.274,Z 333.495,A -85,B 0,C 180,E1 -2151.262,E2 -2151.262} C_VEL
LIN {X 0,Y 704.342,Z 333.494,A -85,B 0,C 180,E1 -2154.052,E2 -2154.052} C_VEL
LIN {X 0,Y 704.28,Z 333.495,A -85,B 0,C 180,E1 -2156.989,E2 -2156.989} C_VEL
LIN {X 0,Y 704.281,Z 333.495,A -85,B 0,C 180,E1 -2159.593,E2 -2159.593} C_VEL
LIN {X 0,Y 704.337,Z 333.489,A -85,B 0,C 180,E1 -2162.522,E2 -2162.522} C_VEL
LIN {X 0,Y 704.273,Z 333.496,A -85,B 0,C 180,E1 -2165.295,E2 -2165.295} C_VEL
LIN {X 0,Y 704.295,Z 333.494,A -85,B 0,C 180,E1 -2167.915,E2 -2167.915} C_VEL
LIN {X 0,Y 704.293,Z 333.489,A -85,B 0,C 180,E1 -2171.05,E2 -2171.05} C_VEL
LIN {X 0,Y 704.272,Z 333.497,A -85,B 0,C 180,E1 -2173.632,E2 -2173.632} C_VEL
LIN {X 0,Y 704.34,Z 333.495,A -85,B 0,C 180,E1 -2176.41,E2 -2176.41} C_VEL
LIN {X 0,Y 704.28,Z 333.49,A -85,B 0,C 180,E1 -2179.317,E2 -2179.317} C_VEL
LIN {X 0,Y 704.277,Z 333.498,A -85,B 0,C 180,E1 -2181.925,E2 -2181.925} C_VEL
LIN {X 0,Y 704.343,Z 333.494,A -85,B 0,C 180,E1 -2184.848,E2 -2184.848} C_VEL
LIN {X 0,Y 704.273,Z 333.494,A -85,B 0,C 180,E1 -2187.662,E2 -2187.662} C_VEL
LIN {X 0,Y 704.292,Z 333.498,A -85,B 0,C 180,E1 -2190.265,E2 -2190.265} C_VEL
LIN {X 0,Y 704.293,Z 333.495,A -85,B 0,C 180,E1 -2193.425,E2 -2193.425} C_VEL
LIN {X 0,Y 704.271,Z 333.498,A -85,B 0,C 180,E1 -2196,E2 -2196} C_VEL
LIN {X 0,Y 704.346,Z 333.498,A -85,B 0,C 180,E1 -2198.863,E2 -2198.863} C_VEL
LIN {X 0,Y 704.278,Z 333.496,A -85,B 0,C 180,E1 -2201.748,E2 -2201.748} C_VEL
LIN {X 0,Y 704.278,Z 333.499,A -85,B 0,C 180,E1 -2204.312,E2 -2204.312} C_VEL
LIN {X 0,Y 704.338,Z 333.493,A -85,B 0,C 180,E1 -2207.267,E2 -2207.267} C_VEL
LIN {X 0,Y 704.272,Z 333.502,A -85,B 0,C 180,E1 -2210.079,E2 -2210.079} C_VEL
LIN {X 0,Y 704.343,Z 333.517,A -85,B 0,C 180,E1 -2210.993,E2 -2210.993} C_VEL
LIN {X 0,Y 710.717,Z 350.76,A -85,B 0,C 180,E1 -2212.673,E2 -2212.673} C_VEL
LIN {X 0,Y 710.234,Z 377.393,A -85,B 0,C 180,E1 -2214.576,E2 -2214.576} C_VEL
LIN {X 0,Y 713.272,Z 390.551,A -85,B 0,C 180,E1 -2214.909,E2 -2214.909} C_VEL
LIN {X 0,Y 711.766,Z 650.872,A -85,B 0,C 180,E1 -2217.914,E2 -2217.914} C_VEL
LIN {X 0,Y 711.095,Z 767.217,A -85,B 0,C 180,E1 -2219.254,E2 -2219.254} C_VEL
LIN {X 0,Y 710.679,Z 792.763,A -85,B 0,C 180,E1 -2219.694,E2 -2219.694} C_VEL
LIN {X 0,Y 710.262,Z 814.452,A -85,B 0,C 180,E1 -2220.205,E2 -2220.205} C_VEL
LIN {X 0,Y 709.764,Z 838.564,A -85,B 0,C 180,E1 -2220.92,E2 -2220.92} C_VEL
LIN {X 0,Y 709.16,Z 860.49,A -85,B 0,C 180,E1 -2221.722,E2 -2221.722} C_VEL
LIN {X 0,Y 708.561,Z 883.171,A -85,B 0,C 180,E1 -2222.702,E2 -2222.702} C_VEL
LIN {X 0,Y 707.876,Z 904.76,A -85,B 0,C 180,E1 -2223.806,E2 -2223.806} C_VEL
LIN {X 0,Y 707.237,Z 925.752,A -85,B 0,C 180,E1 -2225.038,E2 -2225.038} C_VEL
LIN {X 0,Y 706.621,Z 945.052,A -85,B 0,C 180,E1 -2226.349,E2 -2226.349} C_VEL
LIN {X 0,Y 706.067,Z 963.763,A -85,B 0,C 180,E1 -2227.783,E2 -2227.783} C_VEL
LIN {X 0,Y 705.557,Z 980.805,A -85,B 0,C 180,E1 -2229.282,E2 -2229.282} C_VEL
LIN {X 0,Y 705.128,Z 996.967,A -85,B 0,C 180,E1 -2230.879,E2 -2230.879} C_VEL
LIN {X 0,Y 704.773,Z 1011.224,A -85,B 0,C 180,E1 -2232.496,E2 -2232.496} C_VEL
LIN {X 0,Y 704.503,Z 1025.061,A -85,B 0,C 180,E1 -2234.271,E2 -2234.271} C_VEL
LIN {X 0,Y 704.267,Z 1036.798,A -85,B 0,C 180,E1 -2236.033,E2 -2236.033} C_VEL
LIN {X 0,Y 704.122,Z 1046.947,A -85,B 0,C 180,E1 -2237.785,E2 -2237.785} C_VEL
LIN {X 0,Y 704.017,Z 1056.539,A -85,B 0,C 180,E1 -2239.774,E2 -2239.774} C_VEL
LIN {X 0,Y 703.947,Z 1063.12,A -85,B 0,C 180,E1 -2241.423,E2 -2241.423} C_VEL
LIN {X 0,Y 703.913,Z 1069.451,A -85,B 0,C 180,E1 -2243.393,E2 -2243.393} C_VEL
LIN {X 0,Y 703.919,Z 1073.814,A -85,B 0,C 180,E1 -2245.274,E2 -2245.274} C_VEL
LIN {X 0,Y 703.909,Z 1076.797,A -85,B 0,C 180,E1 -2247.15,E2 -2247.15} C_VEL
LIN {X 0,Y 703.902,Z 1078.284,A -85,B 0,C 180,E1 -2249.186,E2 -2249.186} C_VEL
LIN {X 0,Y 703.907,Z 1078.262,A -85,B 0,C 180,E1 -2250.895,E2 -2250.895} C_VEL
LIN {X 0,Y 703.916,Z 1076.573,A -85,B 0,C 180,E1 -2253.013,E2 -2253.013} C_VEL
LIN {X 0,Y 703.919,Z 1073.655,A -85,B 0,C 180,E1 -2254.807,E2 -2254.807} C_VEL
LIN {X 0,Y 703.921,Z 1069.015,A -85,B 0,C 180,E1 -2256.771,E2 -2256.771} C_VEL
LIN {X 0,Y 703.945,Z 1062.815,A -85,B 0,C 180,E1 -2258.66,E2 -2258.66} C_VEL
LIN {X 0,Y 704.025,Z 1056.183,A -85,B 0,C 180,E1 -2260.309,E2 -2260.309} C_VEL
LIN {X 0,Y 704.13,Z 1046.399,A -85,B 0,C 180,E1 -2262.315,E2 -2262.315} C_VEL
LIN {X 0,Y 704.267,Z 1036.8,A -85,B 0,C 180,E1 -2263.967,E2 -2263.967} C_VEL
LIN {X 0,Y 704.511,Z 1024.439,A -85,B 0,C 180,E1 -2265.813,E2 -2265.813} C_VEL
LIN {X 0,Y 704.773,Z 1011.224,A -85,B 0,C 180,E1 -2267.504,E2 -2267.504} C_VEL
LIN {X 0,Y 705.147,Z 996.175,A -85,B 0,C 180,E1 -2269.206,E2 -2269.206} C_VEL
LIN {X 0,Y 705.592,Z 979.534,A -85,B 0,C 180,E1 -2270.836,E2 -2270.836} C_VEL
LIN {X 0,Y 706.116,Z 961.607,A -85,B 0,C 180,E1 -2272.39,E2 -2272.39} C_VEL
LIN {X 0,Y 706.659,Z 944.007,A -85,B 0,C 180,E1 -2273.726,E2 -2273.726} C_VEL
LIN {X 0,Y 707.287,Z 923.622,A -85,B 0,C 180,E1 -2275.094,E2 -2275.094} C_VEL
LIN {X 0,Y 707.908,Z 903.833,A -85,B 0,C 180,E1 -2276.244,E2 -2276.244} C_VEL
LIN {X 0,Y 708.586,Z 882.24,A -85,B 0,C 180,E1 -2277.343,E2 -2277.343} C_VEL
LIN {X 0,Y 709.159,Z 860.493,A -85,B 0,C 180,E1 -2278.278,E2 -2278.278} C_VEL
LIN {X 0,Y 709.764,Z 838.565,A -85,B 0,C 180,E1 -2279.08,E2 -2279.08} C_VEL
LIN {X 0,Y 710.264,Z 814.228,A -85,B 0,C 180,E1 -2279.801,E2 -2279.801} C_VEL
LIN {X 0,Y 710.693,Z 792.376,A -85,B 0,C 180,E1 -2280.314,E2 -2280.314} C_VEL
LIN {X 0,Y 711.097,Z 767.07,A -85,B 0,C 180,E1 -2280.748,E2 -2280.748} C_VEL
LIN {X 0,Y 711.941,Z 619.333,A -85,B 0,C 180,E1 -2282.446,E2 -2282.446} C_VEL
LIN {X 0,Y 713.239,Z 389.492,A -85,B 0,C 180,E1 -2285.106,E2 -2285.106} C_VEL
LIN {X 0,Y 710.16,Z 376.685,A -85,B 0,C 180,E1 -2285.457,E2 -2285.457} C_VEL
LIN {X 0,Y 710.659,Z 350.511,A -85,B 0,C 180,E1 -2287.349,E2 -2287.349} C_VEL
LIN {X 0,Y 704.337,Z 333.5,A -85,B 0,C 180,E1 -2289.039,E2 -2289.039} C_VEL
LIN {X 0,Y 704.27,Z 333.501,A -85,B 0,C 180,E1 -2291.858,E2 -2291.858} C_VEL
LIN {X 0,Y 704.314,Z 333.497,A -85,B 0,C 180,E1 -2294.547,E2 -2294.547} C_VEL
LIN {X 0,Y 704.286,Z 333.5,A -85,B 0,C 180,E1 -2297.595,E2 -2297.595} C_VEL
LIN {X 0,Y 704.272,Z 333.494,A -85,B 0,C 180,E1 -2300.185,E2 -2300.185} C_VEL
LIN {X 0,Y 704.345,Z 333.493,A -85,B 0,C 180,E1 -2303.057,E2 -2303.057} C_VEL
LIN {X 0,Y 704.276,Z 333.496,A -85,B 0,C 180,E1 -2305.889,E2 -2305.889} C_VEL
LIN {X 0,Y 704.281,Z 333.494,A -85,B 0,C 180,E1 -2308.502,E2 -2308.502} C_VEL
LIN {X 0,Y 704.326,Z 333.496,A -85,B 0,C 180,E1 -2311.51,E2 -2311.51} C_VEL
LIN {X 0,Y 704.271,Z 333.496,A -85,B 0,C 180,E1 -2314.25,E2 -2314.25} C_VEL
LIN {X 0,Y 704.329,Z 333.488,A -85,B 0,C 180,E1 -2317.02,E2 -2317.02} C_VEL
LIN {X 0,Y 704.283,Z 333.494,A -85,B 0,C 180,E1 -2320.028,E2 -2320.028} C_VEL
LIN {X 0,Y 704.279,Z 333.495,A -85,B 0,C 180,E1 -2322.654,E2 -2322.654} C_VEL
LIN {X 0,Y 704.343,Z 333.493,A -85,B 0,C 180,E1 -2325.615,E2 -2325.615} C_VEL
LIN {X 0,Y 704.273,Z 333.496,A -85,B 0,C 180,E1 -2328.452,E2 -2328.452} C_VEL
LIN {X 0,Y 704.316,Z 333.487,A -85,B 0,C 180,E1 -2331.18,E2 -2331.18} C_VEL
LIN {X 0,Y 704.288,Z 333.495,A -85,B 0,C 180,E1 -2334.215,E2 -2334.215} C_VEL
LIN {X 0,Y 704.276,Z 333.493,A -85,B 0,C 180,E1 -2336.826,E2 -2336.826} C_VEL
LIN {X 0,Y 704.347,Z 333.496,A -85,B 0,C 180,E1 -2339.756,E2 -2339.756} C_VEL
LIN {X 0,Y 704.275,Z 333.497,A -85,B 0,C 180,E1 -2342.604,E2 -2342.604} C_VEL
LIN {X 0,Y 704.293,Z 333.491,A -85,B 0,C 180,E1 -2345.213,E2 -2345.213} C_VEL
LIN {X 0,Y 704.302,Z 333.499,A -85,B 0,C 180,E1 -2348.326,E2 -2348.326} C_VEL
LIN {X 0,Y 704.273,Z 333.489,A -85,B 0,C 180,E1 -2350.967,E2 -2350.967} C_VEL
LIN {X 0,Y 704.344,Z 333.493,A -85,B 0,C 180,E1 -2353.83,E2 -2353.83} C_VEL
LIN {X 0,Y 704.279,Z 333.495,A -85,B 0,C 180,E1 -2356.751,E2 -2356.751} C_VEL
LIN {X 0,Y 704.29,Z 333.494,A -85,B 0,C 180,E1 -2359.403,E2 -2359.403} C_VEL
LIN {X 0,Y 704.336,Z 333.488,A -85,B 0,C 180,E1 -2361.847,E2 -2361.847} C_VEL
LIN {X 0,Y 703.381,Z 333.617,A -85,B 0,C 180,E1 -2362.473,E2 -2362.473} C_VEL
LIN {X 0,Y 696.926,Z 334.421,A -85,B 0,C 180,E1 -2364.228,E2 -2364.228} C_VEL
LIN {X 0,Y 696.356,Z 334.481,A -85,B 0,C 180,E1 -2364.684,E2 -2364.684} C_VEL
LIN {X 0,Y 696.341,Z 334.484,A -85,B 0,C 180,E1 -2367.355,E2 -2367.355} C_VEL
LIN {X 0,Y 696.407,Z 334.479,A -85,B 0,C 180,E1 -2370.263,E2 -2370.263} C_VEL
LIN {X 0,Y 696.337,Z 334.481,A -85,B 0,C 180,E1 -2373.168,E2 -2373.168} C_VEL
LIN {X 0,Y 696.384,Z 334.482,A -85,B 0,C 180,E1 -2375.963,E2 -2375.963} C_VEL
LIN {X 0,Y 696.349,Z 334.486,A -85,B 0,C 180,E1 -2379.029,E2 -2379.029} C_VEL
LIN {X 0,Y 696.346,Z 334.486,A -85,B 0,C 180,E1 -2381.697,E2 -2381.697} C_VEL
LIN {X 0,Y 696.393,Z 334.471,A -85,B 0,C 180,E1 -2384.713,E2 -2384.713} C_VEL
LIN {X 0,Y 696.339,Z 334.485,A -85,B 0,C 180,E1 -2387.445,E2 -2387.445} C_VEL
LIN {X 0,Y 696.384,Z 334.485,A -85,B 0,C 180,E1 -2390.19,E2 -2390.19} C_VEL
LIN {X 0,Y 696.353,Z 334.493,A -85,B 0,C 180,E1 -2393.248,E2 -2393.248} C_VEL
LIN {X 0,Y 696.422,Z 334.619,A -85,B 0,C 180,E1 -2394.748,E2 -2394.748} C_VEL
LIN {X 0,Y 701.138,Z 347.973,A -85,B 0,C 180,E1 -2396.098,E2 -2396.098} C_VEL
LIN {X 0,Y 704.636,Z 354.675,A -85,B 0,C 180,E1 -2396.386,E2 -2396.386} C_VEL
LIN {X 0,Y 706.663,Z 363.004,A -85,B 0,C 180,E1 -2396.606,E2 -2396.606} C_VEL
LIN {X 0,Y 705.128,Z 598.248,A -85,B 0,C 180,E1 -2399.352,E2 -2399.352} C_VEL
LIN {X 0,Y 704.21,Z 737.177,A -85,B 0,C 180,E1 -2400.965,E2 -2400.965} C_VEL
LIN {X 0,Y 703.751,Z 762.768,A -85,B 0,C 180,E1 -2401.409,E2 -2401.409} C_VEL
LIN {X 0,Y 703.256,Z 784.577,A -85,B 0,C 180,E1 -2401.926,E2 -2401.926} C_VEL
LIN {X 0,Y 702.693,Z 808.39,A -85,B 0,C 180,E1 -2402.638,E2 -2402.638} C_VEL
LIN {X 0,Y 702.015,Z 830.201,A -85,B 0,C 180,E1 -2403.441,E2 -2403.441} C_VEL
LIN {X 0,Y 701.319,Z 852.473,A -85,B 0,C 180,E1 -2404.406,E2 -2404.406} C_VEL
LIN {X 0,Y 700.562,Z 873.84,A -85,B 0,C 180,E1 -2405.505,E2 -2405.505} C_VEL
LIN {X 0,Y 699.805,Z 894.874,A -85,B 0,C 180,E1 -2406.741,E2 -2406.741} C_VEL
LIN {X 0,Y 699.102,Z 914.473,A -85,B 0,C 180,E1 -2408.081,E2 -2408.081} C_VEL
LIN {X 0,Y 698.425,Z 933.56,A -85,B 0,C 180,E1 -2409.554,E2 -2409.554} C_VEL
LIN {X 0,Y 697.838,Z 951.002,A -85,B 0,C 180,E1 -2411.106,E2 -2411.106} C_VEL
LIN {X 0,Y 697.32,Z 967.342,A -85,B 0,C 180,E1 -2412.743,E2 -2412.743} C_VEL
LIN {X 0,Y 696.899,Z 982.046,A -85,B 0,C 180,E1 -2414.437,E2 -2414.437} C_VEL
LIN {X 0,Y 696.566,Z 996.198,A -85,B 0,C 180,E1 -2416.299,E2 -2416.299} C_VEL
LIN {X 0,Y 696.32,Z 1007.726,A -85,B 0,C 180,E1 -2418.066,E2 -2418.066} C_VEL
LIN {X 0,Y 696.141,Z 1018.549,A -85,B 0,C 180,E1 -2419.991,E2 -2419.991} C_VEL
LIN {X 0,Y 696.031,Z 1027.063,A -85,B 0,C 180,E1 -2421.824,E2 -2421.824} C_VEL
LIN {X 0,Y 695.956,Z 1033.838,A -85,B 0,C 180,E1 -2423.566,E2 -2423.566} C_VEL
LIN {X 0,Y 695.923,Z 1040.196,A -85,B 0,C 180,E1 -2425.661,E2 -2425.661} C_VEL
LIN {X 0,Y 695.916,Z 1044.164,A -85,B 0,C 180,E1 -2427.447,E2 -2427.447} C_VEL
LIN {X 0,Y 695.896,Z 1047.103,A -85,B 0,C 180,E1 -2429.424,E2 -2429.424} C_VEL
LIN {X 0,Y 695.895,Z 1048.31,A -85,B 0,C 180,E1 -2431.317,E2 -2431.317} C_VEL
LIN {X 0,Y 695.91,Z 1048.212,A -85,B 0,C 180,E1 -2433.13,E2 -2433.13} C_VEL
LIN {X 0,Y 695.91,Z 1046.435,A -85,B 0,C 180,E1 -2435.193,E2 -2435.193} C_VEL
LIN {X 0,Y 695.91,Z 1043.609,A -85,B 0,C 180,E1 -2436.932,E2 -2436.932} C_VEL
LIN {X 0,Y 695.938,Z 1038.914,A -85,B 0,C 180,E1 -2438.927,E2 -2438.927} C_VEL
LIN {X 0,Y 695.953,Z 1032.963,A -85,B 0,C 180,E1 -2440.765,E2 -2440.765} C_VEL
LIN {X 0,Y 696.045,Z 1026.31,A -85,B 0,C 180,E1 -2442.444,E2 -2442.444} C_VEL
LIN {X 0,Y 696.178,Z 1016.28,A -85,B 0,C 180,E1 -2444.524,E2 -2444.524} C_VEL
LIN {X 0,Y 696.349,Z 1006.27,A -85,B 0,C 180,E1 -2446.26,E2 -2446.26} C_VEL
LIN {X 0,Y 696.617,Z 993.585,A -85,B 0,C 180,E1 -2448.157,E2 -2448.157} C_VEL
LIN {X 0,Y 696.966,Z 980.195,A -85,B 0,C 180,E1 -2449.877,E2 -2449.877} C_VEL
LIN {X 0,Y 697.425,Z 963.824,A -85,B 0,C 180,E1 -2451.715,E2 -2451.715} C_VEL
LIN {X 0,Y 697.931,Z 948.197,A -85,B 0,C 180,E1 -2453.247,E2 -2453.247} C_VEL
LIN {X 0,Y 698.567,Z 929.18,A -85,B 0,C 180,E1 -2454.886,E2 -2454.886} C_VEL
LIN {X 0,Y 699.202,Z 911.507,A -85,B 0,C 180,E1 -2456.224,E2 -2456.224} C_VEL
LIN {X 0,Y 699.962,Z 890.491,A -85,B 0,C 180,E1 -2457.616,E2 -2457.616} C_VEL
LIN {X 0,Y 700.64,Z 871.756,A -85,B 0,C 180,E1 -2458.7,E2 -2458.7} C_VEL
LIN {X 0,Y 701.397,Z 849.133,A -85,B 0,C 180,E1 -2459.836,E2 -2459.836} C_VEL
LIN {X 0,Y 702.059,Z 828.842,A -85,B 0,C 180,E1 -2460.703,E2 -2460.703} C_VEL
LIN {X 0,Y 702.771,Z 806.24,A -85,B 0,C 180,E1 -2461.525,E2 -2461.525} C_VEL
LIN {X 0,Y 703.296,Z 782.52,A -85,B 0,C 180,E1 -2462.218,E2 -2462.218} C_VEL
LIN {X 0,Y 703.893,Z 758.545,A -85,B 0,C 180,E1 -2462.769,E2 -2462.769} C_VEL
LIN {X 0,Y 704.229,Z 734.414,A -85,B 0,C 180,E1 -2463.162,E2 -2463.162} C_VEL
LIN {X 0,Y 705.908,Z 478.384,A -85,B 0,C 180,E1 -2466.127,E2 -2466.127} C_VEL
LIN {X 0,Y 706.499,Z 361.579,A -85,B 0,C 180,E1 -2467.511,E2 -2467.511} C_VEL
LIN {X 0,Y 703.911,Z 352.9,A -85,B 0,C 180,E1 -2467.768,E2 -2467.768} C_VEL
LIN {X 0,Y 700.814,Z 347.209,A -85,B 0,C 180,E1 -2468.041,E2 -2468.041} C_VEL
LIN {X 0,Y 696.408,Z 334.488,A -85,B 0,C 180,E1 -2469.373,E2 -2469.373} C_VEL
LIN {X 0,Y 696.341,Z 334.489,A -85,B 0,C 180,E1 -2472.311,E2 -2472.311} C_VEL
LIN {X 0,Y 696.354,Z 334.487,A -85,B 0,C 180,E1 -2474.948,E2 -2474.948} C_VEL
LIN {X 0,Y 696.367,Z 334.48,A -85,B 0,C 180,E1 -2478.054,E2 -2478.054} C_VEL
LIN {X 0,Y 696.336,Z 334.482,A -85,B 0,C 180,E1 -2480.711,E2 -2480.711} C_VEL
LIN {X 0,Y 696.398,Z 334.472,A -85,B 0,C 180,E1 -2483.528,E2 -2483.528} C_VEL
LIN {X 0,Y 696.347,Z 334.484,A -85,B 0,C 180,E1 -2486.439,E2 -2486.439} C_VEL
LIN {X 0,Y 696.344,Z 334.483,A -85,B 0,C 180,E1 -2489.065,E2 -2489.065} C_VEL
LIN {X 0,Y 696.408,Z 334.481,A -85,B 0,C 180,E1 -2492.007,E2 -2492.007} C_VEL
LIN {X 0,Y 696.335,Z 334.482,A -85,B 0,C 180,E1 -2494.847,E2 -2494.847} C_VEL
LIN {X 0,Y 696.389,Z 334.487,A -85,B 0,C 180,E1 -2497.636,E2 -2497.636} C_VEL
LIN {X 0,Y 696.349,Z 334.483,A -85,B 0,C 180,E1 -2500.629,E2 -2500.629} C_VEL
LIN {X 0,Y 696.342,Z 334.485,A -85,B 0,C 180,E1 -2503.287,E2 -2503.287} C_VEL
LIN {X 0,Y 696.396,Z 334.48,A -85,B 0,C 180,E1 -2506.296,E2 -2506.296} C_VEL
LIN {X 0,Y 696.334,Z 334.484,A -85,B 0,C 180,E1 -2509.074,E2 -2509.074} C_VEL
LIN {X 0,Y 696.381,Z 334.487,A -85,B 0,C 180,E1 -2511.828,E2 -2511.828} C_VEL
LIN {X 0,Y 696.345,Z 334.481,A -85,B 0,C 180,E1 -2514.892,E2 -2514.892} C_VEL
LIN {X 0,Y 696.341,Z 334.487,A -85,B 0,C 180,E1 -2517.531,E2 -2517.531} C_VEL
LIN {X 0,Y 696.404,Z 334.482,A -85,B 0,C 180,E1 -2520.494,E2 -2520.494} C_VEL
LIN {X 0,Y 696.333,Z 334.48,A -85,B 0,C 180,E1 -2523.293,E2 -2523.293} C_VEL
LIN {X 0,Y 696.373,Z 334.489,A -85,B 0,C 180,E1 -2526.017,E2 -2526.017} C_VEL
LIN {X 0,Y 696.348,Z 334.484,A -85,B 0,C 180,E1 -2529.088,E2 -2529.088} C_VEL
LIN {X 0,Y 696.335,Z 334.481,A -85,B 0,C 180,E1 -2531.681,E2 -2531.681} C_VEL
LIN {X 0,Y 696.406,Z 334.478,A -85,B 0,C 180,E1 -2534.598,E2 -2534.598} C_VEL
LIN {X 0,Y 696.335,Z 334.485,A -85,B 0,C 180,E1 -2537.464,E2 -2537.464} C_VEL
LIN {X 0,Y 696.354,Z 334.482,A -85,B 0,C 180,E1 -2540.103,E2 -2540.103} C_VEL
LIN {X 0,Y 696.353,Z 334.479,A -85,B 0,C 180,E1 -2543.258,E2 -2543.258} C_VEL
LIN {X 0,Y 696.335,Z 334.486,A -85,B 0,C 180,E1 -2545.882,E2 -2545.882} C_VEL
LIN {X 0,Y 696.409,Z 334.485,A -85,B 0,C 180,E1 -2548.75,E2 -2548.75} C_VEL
LIN {X 0,Y 696.335,Z 334.485,A -85,B 0,C 180,E1 -2551.624,E2 -2551.624} C_VEL
LIN {X 0,Y 696.346,Z 334.489,A -85,B 0,C 180,E1 -2554.255,E2 -2554.255} C_VEL
LIN {X 0,Y 696.377,Z 334.483,A -85,B 0,C 180,E1 -2557.301,E2 -2557.301} C_VEL
LIN {X 0,Y 696.333,Z 334.487,A -85,B 0,C 180,E1 -2560.039,E2 -2560.039} C_VEL
LIN {X 0,Y 696.399,Z 334.481,A -85,B 0,C 180,E1 -2562.888,E2 -2562.888} C_VEL
LIN {X 0,Y 696.337,Z 334.487,A -85,B 0,C 180,E1 -2565.859,E2 -2565.859} C_VEL
LIN {X 0,Y 696.342,Z 334.491,A -85,B 0,C 180,E1 -2568.441,E2 -2568.441} C_VEL
LIN {X 0,Y 696.357,Z 334.56,A -85,B 0,C 180,E1 -2570.559,E2 -2570.559} C_VEL
LIN {X 0,Y 703.699,Z 354.082,A -85,B 0,C 180,E1 -2572.493,E2 -2572.493} C_VEL
LIN {X 0,Y 703.258,Z 377.512,A -85,B 0,C 180,E1 -2574.173,E2 -2574.173} C_VEL
LIN {X 0,Y 706.709,Z 392.231,A -85,B 0,C 180,E1 -2574.554,E2 -2574.554} C_VEL
LIN {X 0,Y 704.974,Z 652.667,A -85,B 0,C 180,E1 -2577.588,E2 -2577.588} C_VEL
LIN {X 0,Y 704.209,Z 767.356,A -85,B 0,C 180,E1 -2578.922,E2 -2578.922} C_VEL
LIN {X 0,Y 703.745,Z 792.891,A -85,B 0,C 180,E1 -2579.367,E2 -2579.367} C_VEL
LIN {X 0,Y 703.253,Z 814.671,A -85,B 0,C 180,E1 -2579.883,E2 -2579.883} C_VEL
LIN {X 0,Y 702.689,Z 838.561,A -85,B 0,C 180,E1 -2580.599,E2 -2580.599} C_VEL
LIN {X 0,Y 702.044,Z 859.357,A -85,B 0,C 180,E1 -2581.363,E2 -2581.363} C_VEL
LIN {X 0,Y 701.345,Z 881.247,A -85,B 0,C 180,E1 -2582.305,E2 -2582.305} C_VEL
LIN {X 0,Y 700.588,Z 903.141,A -85,B 0,C 180,E1 -2583.421,E2 -2583.421} C_VEL
LIN {X 0,Y 699.874,Z 922.83,A -85,B 0,C 180,E1 -2584.571,E2 -2584.571} C_VEL
LIN {X 0,Y 699.142,Z 943.233,A -85,B 0,C 180,E1 -2585.946,E2 -2585.946} C_VEL
LIN {X 0,Y 698.498,Z 961.254,A -85,B 0,C 180,E1 -2587.324,E2 -2587.324} C_VEL
LIN {X 0,Y 697.901,Z 978.856,A -85,B 0,C 180,E1 -2588.86,E2 -2588.86} C_VEL
LIN {X 0,Y 697.402,Z 994.485,A -85,B 0,C 180,E1 -2590.397,E2 -2590.397} C_VEL
LIN {X 0,Y 696.975,Z 1009.811,A -85,B 0,C 180,E1 -2592.121,E2 -2592.121} C_VEL
LIN {X 0,Y 696.626,Z 1022.853,A -85,B 0,C 180,E1 -2593.79,E2 -2593.79} C_VEL
LIN {X 0,Y 696.344,Z 1036.08,A -85,B 0,C 180,E1 -2595.754,E2 -2595.754} C_VEL
LIN {X 0,Y 696.176,Z 1046.028,A -85,B 0,C 180,E1 -2597.474,E2 -2597.474} C_VEL
LIN {X 0,Y 696.049,Z 1055.829,A -85,B 0,C 180,E1 -2599.488,E2 -2599.488} C_VEL
LIN {X 0,Y 695.954,Z 1062.816,A -85,B 0,C 180,E1 -2601.24,E2 -2601.24} C_VEL
LIN {X 0,Y 695.931,Z 1069.015,A -85,B 0,C 180,E1 -2603.151,E2 -2603.151} C_VEL
LIN {X 0,Y 695.92,Z 1073.656,A -85,B 0,C 180,E1 -2605.137,E2 -2605.137} C_VEL
LIN {X 0,Y 695.916,Z 1076.573,A -85,B 0,C 180,E1 -2606.953,E2 -2606.953} C_VEL
LIN {X 0,Y 695.907,Z 1078.262,A -85,B 0,C 180,E1 -2609.094,E2 -2609.094} C_VEL
LIN {X 0,Y 695.902,Z 1078.284,A -85,B 0,C 180,E1 -2610.823,E2 -2610.823} C_VEL
LIN {X 0,Y 695.91,Z 1076.797,A -85,B 0,C 180,E1 -2612.883,E2 -2612.883} C_VEL
LIN {X 0,Y 695.92,Z 1073.814,A -85,B 0,C 180,E1 -2614.78,E2 -2614.78} C_VEL
LIN {X 0,Y 695.918,Z 1069.451,A -85,B 0,C 180,E1 -2616.683,E2 -2616.683} C_VEL
LIN {X 0,Y 695.953,Z 1063.12,A -85,B 0,C 180,E1 -2618.676,E2 -2618.676} C_VEL
LIN {X 0,Y 696.042,Z 1056.539,A -85,B 0,C 180,E1 -2620.345,E2 -2620.345} C_VEL
LIN {X 0,Y 696.163,Z 1046.947,A -85,B 0,C 180,E1 -2622.357,E2 -2622.357} C_VEL
LIN {X 0,Y 696.329,Z 1036.802,A -85,B 0,C 180,E1 -2624.129,E2 -2624.129} C_VEL
LIN {X 0,Y 696.605,Z 1024.438,A -85,B 0,C 180,E1 -2625.997,E2 -2625.997} C_VEL
LIN {X 0,Y 696.931,Z 1011.226,A -85,B 0,C 180,E1 -2627.707,E2 -2627.707} C_VEL
LIN {X 0,Y 697.354,Z 996.174,A -85,B 0,C 180,E1 -2629.43,E2 -2629.43} C_VEL
LIN {X 0,Y 697.847,Z 980.463,A -85,B 0,C 180,E1 -2630.99,E2 -2630.99} C_VEL
LIN {X 0,Y 698.456,Z 962.713,A -85,B 0,C 180,E1 -2632.561,E2 -2632.561} C_VEL
LIN {X 0,Y 699.099,Z 944.448,A -85,B 0,C 180,E1 -2633.966,E2 -2633.966} C_VEL
LIN {X 0,Y 699.821,Z 924.352,A -85,B 0,C 180,E1 -2635.336,E2 -2635.336} C_VEL
LIN {X 0,Y 700.556,Z 903.948,A -85,B 0,C 180,E1 -2636.535,E2 -2636.535} C_VEL
LIN {X 0,Y 701.324,Z 882.242,A -85,B 0,C 180,E1 -2637.65,E2 -2637.65} C_VEL
LIN {X 0,Y 702.005,Z 860.492,A -85,B 0,C 180,E1 -2638.592,E2 -2638.592} C_VEL
LIN {X 0,Y 702.641,Z 839.846,A -85,B 0,C 180,E1 -2639.356,E2 -2639.356} C_VEL
LIN {X 0,Y 703.252,Z 814.781,A -85,B 0,C 180,E1 -2640.114,E2 -2640.114} C_VEL
LIN {X 0,Y 703.742,Z 793.026,A -85,B 0,C 180,E1 -2640.63,E2 -2640.63} C_VEL
LIN {X 0,Y 704.209,Z 767.542,A -85,B 0,C 180,E1 -2641.075,E2 -2641.075} C_VEL
LIN {X 0,Y 704.904,Z 663.834,A -85,B 0,C 180,E1 -2642.283,E2 -2642.283} C_VEL
LIN {X 0,Y 706.665,Z 398.597,A -85,B 0,C 180,E1 -2645.37,E2 -2645.37} C_VEL
LIN {X 0,Y 706.506,Z 390.587,A -85,B 0,C 180,E1 -2645.477,E2 -2645.477} C_VEL
LIN {X 0,Y 703.158,Z 376.685,A -85,B 0,C 180,E1 -2645.864,E2 -2645.864} C_VEL
LIN {X 0,Y 703.622,Z 353.739,A -85,B 0,C 180,E1 -2647.537,E2 -2647.537} C_VEL
LIN {X 0,Y 696.347,Z 334.498,A -85,B 0,C 180,E1 -2649.462,E2 -2649.462} C_VEL
LIN {X 0,Y 696.335,Z 334.49,A -85,B 0,C 180,E1 -2652.065,E2 -2652.065} C_VEL
LIN {X 0,Y 696.408,Z 334.488,A -85,B 0,C 180,E1 -2654.943,E2 -2654.943} C_VEL
LIN {X 0,Y 696.335,Z 334.489,A -85,B 0,C 180,E1 -2657.812,E2 -2657.812} C_VEL
LIN {X 0,Y 696.351,Z 334.481,A -85,B 0,C 180,E1 -2660.451,E2 -2660.451} C_VEL
LIN {X 0,Y 696.355,Z 334.489,A -85,B 0,C 180,E1 -2663.628,E2 -2663.628} C_VEL
LIN {X 0,Y 696.334,Z 334.483,A -85,B 0,C 180,E1 -2666.243,E2 -2666.243} C_VEL
LIN {X 0,Y 696.406,Z 334.481,A -85,B 0,C 180,E1 -2669.068,E2 -2669.068} C_VEL
LIN {X 0,Y 696.336,Z 334.482,A -85,B 0,C 180,E1 -2672.018,E2 -2672.018} C_VEL
LIN {X 0,Y 696.351,Z 334.483,A -85,B 0,C 180,E1 -2674.666,E2 -2674.666} C_VEL
LIN {X 0,Y 696.36,Z 334.488,A -85,B 0,C 180,E1 -2677.812,E2 -2677.812} C_VEL
LIN {X 0,Y 696.332,Z 334.481,A -85,B 0,C 180,E1 -2680.453,E2 -2680.453} C_VEL
LIN {X 0,Y 696.404,Z 334.483,A -85,B 0,C 180,E1 -2683.312,E2 -2683.312} C_VEL
LIN {X 0,Y 696.339,Z 334.484,A -85,B 0,C 180,E1 -2686.21,E2 -2686.21} C_VEL
LIN {X 0,Y 696.344,Z 334.484,A -85,B 0,C 180,E1 -2688.822,E2 -2688.822} C_VEL
LIN {X 0,Y 696.391,Z 334.487,A -85,B 0,C 180,E1 -2691.828,E2 -2691.828} C_VEL
LIN {X 0,Y 696.335,Z 334.482,A -85,B 0,C 180,E1 -2694.562,E2 -2694.562} C_VEL
LIN {X 0,Y 696.387,Z 334.48,A -85,B 0,C 180,E1 -2697.367,E2 -2697.367} C_VEL
LIN {X 0,Y 696.35,Z 334.479,A -85,B 0,C 180,E1 -2700.329,E2 -2700.329} C_VEL
LIN {X 0,Y 696.339,Z 334.484,A -85,B 0,C 180,E1 -2702.963,E2 -2702.963} C_VEL
LIN {X 0,Y 696.404,Z 334.48,A -85,B 0,C 180,E1 -2705.934,E2 -2705.934} C_VEL
LIN {X 0,Y 696.335,Z 334.486,A -85,B 0,C 180,E1 -2708.755,E2 -2708.755} C_VEL
LIN {X 0,Y 696.377,Z 334.474,A -85,B 0,C 180,E1 -2711.513,E2 -2711.513} C_VEL
LIN {X 0,Y 696.35,Z 334.485,A -85,B 0,C 180,E1 -2714.58,E2 -2714.58} C_VEL
LIN {X 0,Y 696.341,Z 334.482,A -85,B 0,C 180,E1 -2717.206,E2 -2717.206} C_VEL
LIN {X 0,Y 696.407,Z 334.483,A -85,B 0,C 180,E1 -2720.157,E2 -2720.157} C_VEL
LIN {X 0,Y 696.337,Z 334.486,A -85,B 0,C 180,E1 -2723.011,E2 -2723.011} C_VEL
LIN {X 0,Y 696.356,Z 334.481,A -85,B 0,C 180,E1 -2724.684,E2 -2724.684} C_VEL
LIN {X 0,Y 695.32,Z 334.607,A -85,B 0,C 180,E1 -2725.318,E2 -2725.318} C_VEL
LIN {X 0,Y 688.91,Z 335.413,A -85,B 0,C 180,E1 -2727.095,E2 -2727.095} C_VEL
LIN {X 0,Y 688.415,Z 335.473,A -85,B 0,C 180,E1 -2727.556,E2 -2727.556} C_VEL
LIN {X 0,Y 688.427,Z 335.478,A -85,B 0,C 180,E1 -2730.702,E2 -2730.702} C_VEL
LIN {X 0,Y 688.4,Z 335.468,A -85,B 0,C 180,E1 -2733.401,E2 -2733.401} C_VEL
LIN {X 0,Y 688.466,Z 335.473,A -85,B 0,C 180,E1 -2736.339,E2 -2736.339} C_VEL
LIN {X 0,Y 688.401,Z 335.473,A -85,B 0,C 180,E1 -2739.27,E2 -2739.27} C_VEL
LIN {X 0,Y 688.441,Z 335.473,A -85,B 0,C 180,E1 -2742.033,E2 -2742.033} C_VEL
LIN {X 0,Y 688.414,Z 335.469,A -85,B 0,C 180,E1 -2745.098,E2 -2745.098} C_VEL
LIN {X 0,Y 688.408,Z 335.472,A -85,B 0,C 180,E1 -2747.796,E2 -2747.796} C_VEL
LIN {X 0,Y 688.457,Z 335.479,A -85,B 0,C 180,E1 -2750.819,E2 -2750.819} C_VEL
LIN {X 0,Y 688.402,Z 335.482,A -85,B 0,C 180,E1 -2753.657,E2 -2753.657} C_VEL
LIN {X 0,Y 688.464,Z 335.6,A -85,B 0,C 180,E1 -2754.305,E2 -2754.305} C_VEL
LIN {X 0,Y 692.869,Z 347.981,A -85,B 0,C 180,E1 -2755.599,E2 -2755.599} C_VEL
LIN {X 0,Y 698.642,Z 358.523,A -85,B 0,C 180,E1 -2756.081,E2 -2756.081} C_VEL
LIN {X 0,Y 700.126,Z 364.887,A -85,B 0,C 180,E1 -2756.248,E2 -2756.248} C_VEL
LIN {X 0,Y 698.375,Z 600.807,A -85,B 0,C 180,E1 -2759.027,E2 -2759.027} C_VEL
LIN {X 0,Y 697.349,Z 737.279,A -85,B 0,C 180,E1 -2760.626,E2 -2760.626} C_VEL
LIN {X 0,Y 696.842,Z 762.859,A -85,B 0,C 180,E1 -2761.074,E2 -2761.074} C_VEL
LIN {X 0,Y 696.277,Z 784.6,A -85,B 0,C 180,E1 -2761.593,E2 -2761.593} C_VEL
LIN {X 0,Y 695.613,Z 809.119,A -85,B 0,C 180,E1 -2762.336,E2 -2762.336} C_VEL
LIN {X 0,Y 694.904,Z 829.549,A -85,B 0,C 180,E1 -2763.094,E2 -2763.094} C_VEL
LIN {X 0,Y 694.092,Z 852.08,A -85,B 0,C 180,E1 -2764.074,E2 -2764.074} C_VEL
LIN {X 0,Y 693.244,Z 873.505,A -85,B 0,C 180,E1 -2765.183,E2 -2765.183} C_VEL
LIN {X 0,Y 692.427,Z 893.68,A -85,B 0,C 180,E1 -2766.377,E2 -2766.377} C_VEL
LIN {X 0,Y 691.596,Z 913.623,A -85,B 0,C 180,E1 -2767.741,E2 -2767.741} C_VEL
LIN {X 0,Y 690.85,Z 932.283,A -85,B 0,C 180,E1 -2769.187,E2 -2769.187} C_VEL
LIN {X 0,Y 690.186,Z 949.438,A -85,B 0,C 180,E1 -2770.712,E2 -2770.712} C_VEL
LIN {X 0,Y 689.612,Z 965.236,A -85,B 0,C 180,E1 -2772.29,E2 -2772.29} C_VEL
LIN {X 0,Y 689.106,Z 980.853,A -85,B 0,C 180,E1 -2774.083,E2 -2774.083} C_VEL
LIN {X 0,Y 688.706,Z 994.67,A -85,B 0,C 180,E1 -2775.891,E2 -2775.891} C_VEL
LIN {X 0,Y 688.405,Z 1006.847,A -85,B 0,C 180,E1 -2777.757,E2 -2777.757} C_VEL
LIN {X 0,Y 688.205,Z 1017.368,A -85,B 0,C 180,E1 -2779.621,E2 -2779.621} C_VEL
LIN {X 0,Y 688.065,Z 1026.459,A -85,B 0,C 180,E1 -2781.56,E2 -2781.56} C_VEL
LIN {X 0,Y 687.961,Z 1033.322,A -85,B 0,C 180,E1 -2783.323,E2 -2783.323} C_VEL
LIN {X 0,Y 687.929,Z 1039.568,A -85,B 0,C 180,E1 -2785.331,E2 -2785.331} C_VEL
LIN {X 0,Y 687.911,Z 1043.735,A -85,B 0,C 180,E1 -2787.167,E2 -2787.167} C_VEL
LIN {X 0,Y 687.912,Z 1046.513,A -85,B 0,C 180,E1 -2788.917,E2 -2788.917} C_VEL
LIN {X 0,Y 687.913,Z 1048.226,A -85,B 0,C 180,E1 -2790.999,E2 -2790.999} C_VEL
LIN {X 0,Y 687.901,Z 1048.296,A -85,B 0,C 180,E1 -2792.833,E2 -2792.833} C_VEL
LIN {X 0,Y 687.899,Z 1046.967,A -85,B 0,C 180,E1 -2794.836,E2 -2794.836} C_VEL
LIN {X 0,Y 687.914,Z 1044.042,A -85,B 0,C 180,E1 -2796.761,E2 -2796.761} C_VEL
LIN {X 0,Y 687.924,Z 1040.142,A -85,B 0,C 180,E1 -2798.526,E2 -2798.526} C_VEL
LIN {X 0,Y 687.96,Z 1033.791,A -85,B 0,C 180,E1 -2800.637,E2 -2800.637} C_VEL
LIN {X 0,Y 688.058,Z 1026.922,A -85,B 0,C 180,E1 -2802.42,E2 -2802.42} C_VEL
LIN {X 0,Y 688.197,Z 1017.816,A -85,B 0,C 180,E1 -2804.386,E2 -2804.386} C_VEL
LIN {X 0,Y 688.398,Z 1007.167,A -85,B 0,C 180,E1 -2806.28,E2 -2806.28} C_VEL
LIN {X 0,Y 688.704,Z 994.743,A -85,B 0,C 180,E1 -2808.189,E2 -2808.189} C_VEL
LIN {X 0,Y 689.089,Z 981.417,A -85,B 0,C 180,E1 -2809.937,E2 -2809.937} C_VEL
LIN {X 0,Y 689.58,Z 966.197,A -85,B 0,C 180,E1 -2811.7,E2 -2811.7} C_VEL
LIN {X 0,Y 690.172,Z 949.803,A -85,B 0,C 180,E1 -2813.343,E2 -2813.343} C_VEL
LIN {X 0,Y 690.854,Z 932.213,A -85,B 0,C 180,E1 -2814.909,E2 -2814.909} C_VEL
LIN {X 0,Y 691.597,Z 913.611,A -85,B 0,C 180,E1 -2816.35,E2 -2816.35} C_VEL
LIN {X 0,Y 692.455,Z 893.015,A -85,B 0,C 180,E1 -2817.754,E2 -2817.754} C_VEL
LIN {X 0,Y 693.237,Z 873.73,A -85,B 0,C 180,E1 -2818.895,E2 -2818.895} C_VEL
LIN {X 0,Y 694.099,Z 851.82,A -85,B 0,C 180,E1 -2820.028,E2 -2820.028} C_VEL
LIN {X 0,Y 694.886,Z 830.038,A -85,B 0,C 180,E1 -2820.977,E2 -2820.977} C_VEL
LIN {X 0,Y 695.629,Z 808.789,A -85,B 0,C 180,E1 -2821.766,E2 -2821.766} C_VEL
LIN {X 0,Y 696.285,Z 784.259,A -85,B 0,C 180,E1 -2822.506,E2 -2822.506} C_VEL
LIN {X 0,Y 696.859,Z 762.366,A -85,B 0,C 180,E1 -2823.026,E2 -2823.026} C_VEL
LIN {X 0,Y 697.352,Z 737.001,A -85,B 0,C 180,E1 -2823.468,E2 -2823.468} C_VEL
LIN {X 0,Y 699.01,Z 511.807,A -85,B 0,C 180,E1 -2826.104,E2 -2826.104} C_VEL
LIN {X 0,Y 699.971,Z 363.45,A -85,B 0,C 180,E1 -2827.869,E2 -2827.869} C_VEL
LIN {X 0,Y 697.936,Z 356.872,A -85,B 0,C 180,E1 -2828.072,E2 -2828.072} C_VEL
LIN {X 0,Y 692.659,Z 347.51,A -85,B 0,C 180,E1 -2828.518,E2 -2828.518} C_VEL
LIN {X 0,Y 688.441,Z 335.478,A -85,B 0,C 180,E1 -2829.83,E2 -2829.83} C_VEL
LIN {X 0,Y 688.4,Z 335.479,A -85,B 0,C 180,E1 -2832.599,E2 -2832.599} C_VEL
LIN {X 0,Y 688.466,Z 335.473,A -85,B 0,C 180,E1 -2835.488,E2 -2835.488} C_VEL
LIN {X 0,Y 688.4,Z 335.47,A -85,B 0,C 180,E1 -2838.42,E2 -2838.42} C_VEL
LIN {X 0,Y 688.422,Z 335.474,A -85,B 0,C 180,E1 -2841.137,E2 -2841.137} C_VEL
LIN {X 0,Y 688.415,Z 335.457,A -85,B 0,C 180,E1 -2844.284,E2 -2844.284} C_VEL
LIN {X 0,Y 688.404,Z 335.476,A -85,B 0,C 180,E1 -2846.997,E2 -2846.997} C_VEL
LIN {X 0,Y 688.461,Z 335.471,A -85,B 0,C 180,E1 -2850.026,E2 -2850.026} C_VEL
LIN {X 0,Y 688.398,Z 335.475,A -85,B 0,C 180,E1 -2852.865,E2 -2852.865} C_VEL
LIN {X 0,Y 688.464,Z 335.474,A -85,B 0,C 180,E1 -2855.731,E2 -2855.731} C_VEL
LIN {X 0,Y 688.403,Z 335.47,A -85,B 0,C 180,E1 -2858.708,E2 -2858.708} C_VEL
LIN {X 0,Y 688.411,Z 335.476,A -85,B 0,C 180,E1 -2861.365,E2 -2861.365} C_VEL
LIN {X 0,Y 688.427,Z 335.471,A -85,B 0,C 180,E1 -2864.499,E2 -2864.499} C_VEL
LIN {X 0,Y 688.396,Z 335.473,A -85,B 0,C 180,E1 -2867.16,E2 -2867.16} C_VEL
LIN {X 0,Y 688.465,Z 335.47,A -85,B 0,C 180,E1 -2870.048,E2 -2870.048} C_VEL
LIN {X 0,Y 688.401,Z 335.473,A -85,B 0,C 180,E1 -2872.992,E2 -2872.992} C_VEL
LIN {X 0,Y 688.415,Z 335.474,A -85,B 0,C 180,E1 -2875.668,E2 -2875.668} C_VEL
LIN {X 0,Y 688.417,Z 335.468,A -85,B 0,C 180,E1 -2878.835,E2 -2878.835} C_VEL
LIN {X 0,Y 688.398,Z 335.475,A -85,B 0,C 180,E1 -2881.498,E2 -2881.498} C_VEL
LIN {X 0,Y 688.467,Z 335.474,A -85,B 0,C 180,E1 -2884.415,E2 -2884.415} C_VEL
LIN {X 0,Y 688.396,Z 335.467,A -85,B 0,C 180,E1 -2887.26,E2 -2887.26} C_VEL
LIN {X 0,Y 688.412,Z 335.477,A -85,B 0,C 180,E1 -2889.869,E2 -2889.869} C_VEL
LIN {X 0,Y 688.423,Z 335.472,A -85,B 0,C 180,E1 -2893.01,E2 -2893.01} C_VEL
LIN {X 0,Y 688.394,Z 335.469,A -85,B 0,C 180,E1 -2895.674,E2 -2895.674} C_VEL
LIN {X 0,Y 688.466,Z 335.469,A -85,B 0,C 180,E1 -2898.546,E2 -2898.546} C_VEL
LIN {X 0,Y 688.399,Z 335.474,A -85,B 0,C 180,E1 -2901.471,E2 -2901.471} C_VEL
LIN {X 0,Y 688.408,Z 335.471,A -85,B 0,C 180,E1 -2904.088,E2 -2904.088} C_VEL
LIN {X 0,Y 688.437,Z 335.469,A -85,B 0,C 180,E1 -2907.133,E2 -2907.133} C_VEL
LIN {X 0,Y 688.393,Z 335.474,A -85,B 0,C 180,E1 -2909.786,E2 -2909.786} C_VEL
LIN {X 0,Y 688.439,Z 335.478,A -85,B 0,C 180,E1 -2912.506,E2 -2912.506} C_VEL
LIN {X 0,Y 688.407,Z 335.474,A -85,B 0,C 180,E1 -2915.572,E2 -2915.572} C_VEL
LIN {X 0,Y 688.401,Z 335.476,A -85,B 0,C 180,E1 -2918.226,E2 -2918.226} C_VEL
LIN {X 0,Y 688.454,Z 335.472,A -85,B 0,C 180,E1 -2921.253,E2 -2921.253} C_VEL
LIN {X 0,Y 688.393,Z 335.476,A -85,B 0,C 180,E1 -2924.087,E2 -2924.087} C_VEL
LIN {X 0,Y 688.46,Z 335.472,A -85,B 0,C 180,E1 -2926.952,E2 -2926.952} C_VEL
LIN {X 0,Y 688.404,Z 335.481,A -85,B 0,C 180,E1 -2929.842,E2 -2929.842} C_VEL
LIN {X 0,Y 688.407,Z 335.577,A -85,B 0,C 180,E1 -2930.113,E2 -2930.113} C_VEL
LIN {X 0,Y 696.632,Z 357.318,A -85,B 0,C 180,E1 -2932.306,E2 -2932.306} C_VEL
LIN {X 0,Y 696.264,Z 377.414,A -85,B 0,C 180,E1 -2933.755,E2 -2933.755} C_VEL
LIN {X 0,Y 700.173,Z 394.081,A -85,B 0,C 180,E1 -2934.196,E2 -2934.196} C_VEL
LIN {X 0,Y 698.195,Z 655.721,A -85,B 0,C 180,E1 -2937.271,E2 -2937.271} C_VEL
LIN {X 0,Y 697.347,Z 767.4,A -85,B 0,C 180,E1 -2938.583,E2 -2938.583} C_VEL
LIN {X 0,Y 696.839,Z 792.889,A -85,B 0,C 180,E1 -2939.03,E2 -2939.03} C_VEL
LIN {X 0,Y 696.274,Z 814.669,A -85,B 0,C 180,E1 -2939.55,E2 -2939.55} C_VEL
LIN {X 0,Y 695.638,Z 838.557,A -85,B 0,C 180,E1 -2940.271,E2 -2940.271} C_VEL
LIN {X 0,Y 694.912,Z 859.353,A -85,B 0,C 180,E1 -2941.041,E2 -2941.041} C_VEL
LIN {X 0,Y 694.117,Z 881.251,A -85,B 0,C 180,E1 -2941.991,E2 -2941.991} C_VEL
LIN {X 0,Y 693.26,Z 903.137,A -85,B 0,C 180,E1 -2943.118,E2 -2943.118} C_VEL
LIN {X 0,Y 692.485,Z 922.179,A -85,B 0,C 180,E1 -2944.239,E2 -2944.239} C_VEL
LIN {X 0,Y 691.611,Z 943.23,A -85,B 0,C 180,E1 -2945.667,E2 -2945.667} C_VEL
LIN {X 0,Y 690.896,Z 961.056,A -85,B 0,C 180,E1 -2947.044,E2 -2947.044} C_VEL
LIN {X 0,Y 690.21,Z 978.605,A -85,B 0,C 180,E1 -2948.588,E2 -2948.588} C_VEL
LIN {X 0,Y 689.671,Z 993.638,A -85,B 0,C 180,E1 -2950.08,E2 -2950.08} C_VEL
LIN {X 0,Y 689.135,Z 1009.813,A -85,B 0,C 180,E1 -2951.911,E2 -2951.911} C_VEL
LIN {X 0,Y 688.749,Z 1022.529,A -85,B 0,C 180,E1 -2953.555,E2 -2953.555} C_VEL
LIN {X 0,Y 688.429,Z 1035.761,A -85,B 0,C 180,E1 -2955.533,E2 -2955.533} C_VEL
LIN {X 0,Y 688.229,Z 1045.568,A -85,B 0,C 180,E1 -2957.242,E2 -2957.242} C_VEL
LIN {X 0,Y 688.07,Z 1055.475,A -85,B 0,C 180,E1 -2959.28,E2 -2959.28} C_VEL
LIN {X 0,Y 687.974,Z 1062.513,A -85,B 0,C 180,E1 -2961.053,E2 -2961.053} C_VEL
LIN {X 0,Y 687.953,Z 1068.507,A -85,B 0,C 180,E1 -2962.903,E2 -2962.903} C_VEL
LIN {X 0,Y 687.923,Z 1073.497,A -85,B 0,C 180,E1 -2964.997,E2 -2964.997} C_VEL
LIN {X 0,Y 687.916,Z 1076.461,A -85,B 0,C 180,E1 -2966.834,E2 -2966.834} C_VEL
LIN {X 0,Y 687.914,Z 1078.239,A -85,B 0,C 180,E1 -2969.001,E2 -2969.001} C_VEL
LIN {X 0,Y 687.898,Z 1078.306,A -85,B 0,C 180,E1 -2970.75,E2 -2970.75} C_VEL
LIN {X 0,Y 687.907,Z 1077.017,A -85,B 0,C 180,E1 -2972.749,E2 -2972.749} C_VEL
LIN {X 0,Y 687.92,Z 1073.973,A -85,B 0,C 180,E1 -2974.752,E2 -2974.752} C_VEL
LIN {X 0,Y 687.916,Z 1070.07,A -85,B 0,C 180,E1 -2976.51,E2 -2976.51} C_VEL
LIN {X 0,Y 687.961,Z 1063.726,A -85,B 0,C 180,E1 -2978.61,E2 -2978.61} C_VEL
LIN {X 0,Y 688.057,Z 1056.895,A -85,B 0,C 180,E1 -2980.381,E2 -2980.381} C_VEL
LIN {X 0,Y 688.19,Z 1047.863,A -85,B 0,C 180,E1 -2982.332,E2 -2982.332} C_VEL
LIN {X 0,Y 688.386,Z 1037.323,A -85,B 0,C 180,E1 -2984.21,E2 -2984.21} C_VEL
LIN {X 0,Y 688.696,Z 1025.063,A -85,B 0,C 180,E1 -2986.099,E2 -2986.099} C_VEL
LIN {X 0,Y 689.094,Z 1011.228,A -85,B 0,C 180,E1 -2987.916,E2 -2987.916} C_VEL
LIN {X 0,Y 689.579,Z 996.173,A -85,B 0,C 180,E1 -2989.658,E2 -2989.658} C_VEL
LIN {X 0,Y 690.14,Z 980.462,A -85,B 0,C 180,E1 -2991.236,E2 -2991.236} C_VEL
LIN {X 0,Y 690.837,Z 962.713,A -85,B 0,C 180,E1 -2992.823,E2 -2992.823} C_VEL
LIN {X 0,Y 691.588,Z 943.837,A -85,B 0,C 180,E1 -2994.288,E2 -2994.288} C_VEL
LIN {X 0,Y 692.427,Z 923.628,A -85,B 0,C 180,E1 -2995.671,E2 -2995.671} C_VEL
LIN {X 0,Y 693.227,Z 903.944,A -85,B 0,C 180,E1 -2996.837,E2 -2996.837} C_VEL
LIN {X 0,Y 694.09,Z 882.148,A -85,B 0,C 180,E1 -2997.968,E2 -2997.968} C_VEL
LIN {X 0,Y 694.871,Z 860.488,A -85,B 0,C 180,E1 -2998.914,E2 -2998.914} C_VEL
LIN {X 0,Y 695.586,Z 839.842,A -85,B 0,C 180,E1 -2999.684,E2 -2999.684} C_VEL
LIN {X 0,Y 696.272,Z 814.781,A -85,B 0,C 180,E1 -3000.448,E2 -3000.448} C_VEL
LIN {X 0,Y 696.834,Z 793.024,A -85,B 0,C 180,E1 -3000.967,E2 -3000.967} C_VEL
LIN {X 0,Y 697.348,Z 767.543,A -85,B 0,C 180,E1 -3001.415,E2 -3001.415} C_VEL
LIN {X 0,Y 698.179,Z 657.887,A -85,B 0,C 180,E1 -3002.704,E2 -3002.704} C_VEL
LIN {X 0,Y 700.161,Z 395.555,A -85,B 0,C 180,E1 -3005.787,E2 -3005.787} C_VEL
LIN {X 0,Y 699.898,Z 392.055,A -85,B 0,C 180,E1 -3005.846,E2 -3005.846} C_VEL
LIN {X 0,Y 696.185,Z 376.671,A -85,B 0,C 180,E1 -3006.28,E2 -3006.28} C_VEL
LIN {X 0,Y 696.517,Z 357.059,A -85,B 0,C 180,E1 -3007.721,E2 -3007.721} C_VEL
LIN {X 0,Y 689.28,Z 338.267,A -85,B 0,C 180,E1 -3009.62,E2 -3009.62} C_VEL
LIN {X 0,Y 688.395,Z 335.489,A -85,B 0,C 180,E1 -3009.922,E2 -3009.922} C_VEL
LIN {X 0,Y 688.457,Z 335.476,A -85,B 0,C 180,E1 -3012.707,E2 -3012.707} C_VEL
LIN {X 0,Y 688.401,Z 335.479,A -85,B 0,C 180,E1 -3015.681,E2 -3015.681} C_VEL
LIN {X 0,Y 688.404,Z 335.476,A -85,B 0,C 180,E1 -3018.299,E2 -3018.299} C_VEL
LIN {X 0,Y 688.446,Z 335.478,A -85,B 0,C 180,E1 -3021.352,E2 -3021.352} C_VEL
LIN {X 0,Y 688.395,Z 335.476,A -85,B 0,C 180,E1 -3024.144,E2 -3024.144} C_VEL
LIN {X 0,Y 688.464,Z 335.47,A -85,B 0,C 180,E1 -3027,E2 -3027} C_VEL
LIN {X 0,Y 688.4,Z 335.475,A -85,B 0,C 180,E1 -3029.96,E2 -3029.96} C_VEL
LIN {X 0,Y 688.408,Z 335.468,A -85,B 0,C 180,E1 -3032.585,E2 -3032.585} C_VEL
LIN {X 0,Y 688.438,Z 335.472,A -85,B 0,C 180,E1 -3035.639,E2 -3035.639} C_VEL
LIN {X 0,Y 688.394,Z 335.474,A -85,B 0,C 180,E1 -3038.372,E2 -3038.372} C_VEL
LIN {X 0,Y 688.466,Z 335.466,A -85,B 0,C 180,E1 -3041.25,E2 -3041.25} C_VEL
LIN {X 0,Y 688.4,Z 335.473,A -85,B 0,C 180,E1 -3044.24,E2 -3044.24} C_VEL
LIN {X 0,Y 688.414,Z 335.469,A -85,B 0,C 180,E1 -3046.904,E2 -3046.904} C_VEL
LIN {X 0,Y 688.42,Z 335.469,A -85,B 0,C 180,E1 -3050.047,E2 -3050.047} C_VEL
LIN {X 0,Y 688.398,Z 335.474,A -85,B 0,C 180,E1 -3052.74,E2 -3052.74} C_VEL
LIN {X 0,Y 688.465,Z 335.467,A -85,B 0,C 180,E1 -3055.669,E2 -3055.669} C_VEL
LIN {X 0,Y 688.397,Z 335.474,A -85,B 0,C 180,E1 -3058.585,E2 -3058.585} C_VEL
LIN {X 0,Y 688.436,Z 335.462,A -85,B 0,C 180,E1 -3061.332,E2 -3061.332} C_VEL
LIN {X 0,Y 688.41,Z 335.473,A -85,B 0,C 180,E1 -3064.415,E2 -3064.415} C_VEL
LIN {X 0,Y 688.404,Z 335.469,A -85,B 0,C 180,E1 -3067.092,E2 -3067.092} C_VEL
LIN {X 0,Y 688.452,Z 335.47,A -85,B 0,C 180,E1 -3070.122,E2 -3070.122} C_VEL
LIN {X 0,Y 688.398,Z 335.474,A -85,B 0,C 180,E1 -3072.937,E2 -3072.937} C_VEL
LIN {X 0,Y 688.461,Z 335.468,A -85,B 0,C 180,E1 -3075.759,E2 -3075.759} C_VEL
LIN {X 0,Y 688.406,Z 335.476,A -85,B 0,C 180,E1 -3078.736,E2 -3078.736} C_VEL
LIN {X 0,Y 688.411,Z 335.466,A -85,B 0,C 180,E1 -3081.405,E2 -3081.405} C_VEL
LIN {X 0,Y 688.444,Z 335.471,A -85,B 0,C 180,E1 -3084.452,E2 -3084.452} C_VEL
LIN {X 0,Y 688.399,Z 335.474,A -85,B 0,C 180,E1 -3087.228,E2 -3087.228} C_VEL
LIN {X 0,Y 688.415,Z 335.473,A -85,B 0,C 180,E1 -3087.556,E2 -3087.556} C_VEL
LIN {X 0,Y 687.487,Z 335.597,A -85,B 0,C 180,E1 -3088.197,E2 -3088.197} C_VEL
LIN {X 0,Y 681.003,Z 336.394,A -85,B 0,C 180,E1 -3090.04,E2 -3090.04} C_VEL
LIN {X 0,Y 680.52,Z 336.461,A -85,B 0,C 180,E1 -3090.461,E2 -3090.461} C_VEL
LIN {X 0,Y 680.46,Z 336.458,A -85,B 0,C 180,E1 -3093.269,E2 -3093.269} C_VEL
LIN {X 0,Y 680.521,Z 336.46,A -85,B 0,C 180,E1 -3096.1,E2 -3096.1} C_VEL
LIN {X 0,Y 680.467,Z 336.463,A -85,B 0,C 180,E1 -3099.118,E2 -3099.118} C_VEL
LIN {X 0,Y 680.481,Z 336.464,A -85,B 0,C 180,E1 -3101.844,E2 -3101.844} C_VEL
LIN {X 0,Y 680.479,Z 336.453,A -85,B 0,C 180,E1 -3105.027,E2 -3105.027} C_VEL
LIN {X 0,Y 680.465,Z 336.461,A -85,B 0,C 180,E1 -3107.701,E2 -3107.701} C_VEL
LIN {X 0,Y 680.531,Z 336.465,A -85,B 0,C 180,E1 -3110.61,E2 -3110.61} C_VEL
LIN {X 0,Y 680.464,Z 336.472,A -85,B 0,C 180,E1 -3113.493,E2 -3113.493} C_VEL
LIN {X 0,Y 680.495,Z 336.659,A -85,B 0,C 180,E1 -3113.852,E2 -3113.852} C_VEL
LIN {X 0,Y 684.717,Z 348.244,A -85,B 0,C 180,E1 -3115.094,E2 -3115.094} C_VEL
LIN {X 0,Y 692.718,Z 362.495,A -85,B 0,C 180,E1 -3115.773,E2 -3115.773} C_VEL
LIN {X 0,Y 693.619,Z 366.874,A -85,B 0,C 180,E1 -3115.884,E2 -3115.884} C_VEL
LIN {X 0,Y 691.647,Z 602.962,A -85,B 0,C 180,E1 -3118.69,E2 -3118.69} C_VEL
LIN {X 0,Y 690.512,Z 737.314,A -85,B 0,C 180,E1 -3120.279,E2 -3120.279} C_VEL
LIN {X 0,Y 689.962,Z 762.768,A -85,B 0,C 180,E1 -3120.729,E2 -3120.729} C_VEL
LIN {X 0,Y 689.334,Z 784.408,A -85,B 0,C 180,E1 -3121.248,E2 -3121.248} C_VEL
LIN {X 0,Y 688.597,Z 808.779,A -85,B 0,C 180,E1 -3121.99,E2 -3121.99} C_VEL
LIN {X 0,Y 687.812,Z 829.079,A -85,B 0,C 180,E1 -3122.747,E2 -3122.747} C_VEL
LIN {X 0,Y 686.937,Z 850.775,A -85,B 0,C 180,E1 -3123.694,E2 -3123.694} C_VEL
LIN {X 0,Y 685.975,Z 872.371,A -85,B 0,C 180,E1 -3124.81,E2 -3124.81} C_VEL
LIN {X 0,Y 685.133,Z 891.237,A -85,B 0,C 180,E1 -3125.927,E2 -3125.927} C_VEL
LIN {X 0,Y 684.11,Z 912.774,A -85,B 0,C 180,E1 -3127.394,E2 -3127.394} C_VEL
LIN {X 0,Y 683.33,Z 930.395,A -85,B 0,C 180,E1 -3128.765,E2 -3128.765} C_VEL
LIN {X 0,Y 682.514,Z 948.792,A -85,B 0,C 180,E1 -3130.398,E2 -3130.398} C_VEL
LIN {X 0,Y 681.886,Z 964.475,A -85,B 0,C 180,E1 -3131.977,E2 -3131.977} C_VEL
LIN {X 0,Y 681.282,Z 980.36,A -85,B 0,C 180,E1 -3133.808,E2 -3133.808} C_VEL
LIN {X 0,Y 680.848,Z 993.532,A -85,B 0,C 180,E1 -3135.543,E2 -3135.543} C_VEL
LIN {X 0,Y 680.49,Z 1006.483,A -85,B 0,C 180,E1 -3137.526,E2 -3137.526} C_VEL
LIN {X 0,Y 680.261,Z 1016.589,A -85,B 0,C 180,E1 -3139.327,E2 -3139.327} C_VEL
LIN {X 0,Y 680.076,Z 1026.209,A -85,B 0,C 180,E1 -3141.375,E2 -3141.375} C_VEL
LIN {X 0,Y 679.984,Z 1032.805,A -85,B 0,C 180,E1 -3143.075,E2 -3143.075} C_VEL
LIN {X 0,Y 679.948,Z 1038.981,A -85,B 0,C 180,E1 -3145.023,E2 -3145.023} C_VEL
LIN {X 0,Y 679.915,Z 1043.623,A -85,B 0,C 180,E1 -3147.05,E2 -3147.05} C_VEL
LIN {X 0,Y 679.91,Z 1046.433,A -85,B 0,C 180,E1 -3148.82,E2 -3148.82} C_VEL
LIN {X 0,Y 679.913,Z 1048.21,A -85,B 0,C 180,E1 -3150.927,E2 -3150.927} C_VEL
LIN {X 0,Y 679.899,Z 1048.312,A -85,B 0,C 180,E1 -3152.782,E2 -3152.782} C_VEL
LIN {X 0,Y 679.898,Z 1047.036,A -85,B 0,C 180,E1 -3154.809,E2 -3154.809} C_VEL
LIN {X 0,Y 679.915,Z 1044.156,A -85,B 0,C 180,E1 -3156.756,E2 -3156.756} C_VEL
LIN {X 0,Y 679.926,Z 1040.289,A -85,B 0,C 180,E1 -3158.542,E2 -3158.542} C_VEL
LIN {X 0,Y 679.968,Z 1034.312,A -85,B 0,C 180,E1 -3160.592,E2 -3160.592} C_VEL
LIN {X 0,Y 680.075,Z 1027.177,A -85,B 0,C 180,E1 -3162.482,E2 -3162.482} C_VEL
LIN {X 0,Y 680.233,Z 1018.137,A -85,B 0,C 180,E1 -3164.471,E2 -3164.471} C_VEL
LIN {X 0,Y 680.46,Z 1007.539,A -85,B 0,C 180,E1 -3166.387,E2 -3166.387} C_VEL
LIN {X 0,Y 680.784,Z 995.77,A -85,B 0,C 180,E1 -3168.23,E2 -3168.23} C_VEL
LIN {X 0,Y 681.237,Z 981.917,A -85,B 0,C 180,E1 -3170.088,E2 -3170.088} C_VEL
LIN {X 0,Y 681.793,Z 966.772,A -85,B 0,C 180,E1 -3171.87,E2 -3171.87} C_VEL
LIN {X 0,Y 682.45,Z 950.464,A -85,B 0,C 180,E1 -3173.531,E2 -3173.531} C_VEL
LIN {X 0,Y 683.237,Z 932.67,A -85,B 0,C 180,E1 -3175.141,E2 -3175.141} C_VEL
LIN {X 0,Y 684.068,Z 913.872,A -85,B 0,C 180,E1 -3176.615,E2 -3176.615} C_VEL
LIN {X 0,Y 685.043,Z 893.323,A -85,B 0,C 180,E1 -3178.034,E2 -3178.034} C_VEL
LIN {X 0,Y 685.942,Z 873.257,A -85,B 0,C 180,E1 -3179.231,E2 -3179.231} C_VEL
LIN {X 0,Y 686.886,Z 852.005,A -85,B 0,C 180,E1 -3180.34,E2 -3180.34} C_VEL
LIN {X 0,Y 687.783,Z 829.798,A -85,B 0,C 180,E1 -3181.314,E2 -3181.314} C_VEL
LIN {X 0,Y 688.576,Z 809.336,A -85,B 0,C 180,E1 -3182.08,E2 -3182.08} C_VEL
LIN {X 0,Y 689.331,Z 784.564,A -85,B 0,C 180,E1 -3182.838,E2 -3182.838} C_VEL
LIN {X 0,Y 689.959,Z 762.87,A -85,B 0,C 180,E1 -3183.359,E2 -3183.359} C_VEL
LIN {X 0,Y 690.513,Z 737.402,A -85,B 0,C 180,E1 -3183.809,E2 -3183.809} C_VEL
LIN {X 0,Y 691.622,Z 606.026,A -85,B 0,C 180,E1 -3185.364,E2 -3185.364} C_VEL
LIN {X 0,Y 693.584,Z 370.527,A -85,B 0,C 180,E1 -3188.163,E2 -3188.163} C_VEL
LIN {X 0,Y 693.423,Z 365.152,A -85,B 0,C 180,E1 -3188.24,E2 -3188.24} C_VEL
LIN {X 0,Y 692.074,Z 361.063,A -85,B 0,C 180,E1 -3188.374,E2 -3188.374} C_VEL
LIN {X 0,Y 684.501,Z 347.835,A -85,B 0,C 180,E1 -3189.02,E2 -3189.02} C_VEL
LIN {X 0,Y 680.464,Z 336.47,A -85,B 0,C 180,E1 -3190.282,E2 -3190.282} C_VEL
LIN {X 0,Y 680.482,Z 336.466,A -85,B 0,C 180,E1 -3192.984,E2 -3192.984} C_VEL
LIN {X 0,Y 680.484,Z 336.46,A -85,B 0,C 180,E1 -3196.088,E2 -3196.088} C_VEL
LIN {X 0,Y 680.46,Z 336.458,A -85,B 0,C 180,E1 -3198.794,E2 -3198.794} C_VEL
LIN {X 0,Y 680.529,Z 336.462,A -85,B 0,C 180,E1 -3201.683,E2 -3201.683} C_VEL
LIN {X 0,Y 680.457,Z 336.446,A -85,B 0,C 180,E1 -3204.641,E2 -3204.641} C_VEL
LIN {X 0,Y 680.499,Z 336.467,A -85,B 0,C 180,E1 -3207.367,E2 -3207.367} C_VEL
LIN {X 0,Y 680.472,Z 336.462,A -85,B 0,C 180,E1 -3210.446,E2 -3210.446} C_VEL
LIN {X 0,Y 680.467,Z 336.465,A -85,B 0,C 180,E1 -3213.118,E2 -3213.118} C_VEL
LIN {X 0,Y 680.514,Z 336.461,A -85,B 0,C 180,E1 -3216.167,E2 -3216.167} C_VEL
LIN {X 0,Y 680.458,Z 336.46,A -85,B 0,C 180,E1 -3218.989,E2 -3218.989} C_VEL
LIN {X 0,Y 680.523,Z 336.459,A -85,B 0,C 180,E1 -3221.851,E2 -3221.851} C_VEL
LIN {X 0,Y 680.461,Z 336.462,A -85,B 0,C 180,E1 -3224.837,E2 -3224.837} C_VEL
LIN {X 0,Y 680.476,Z 336.464,A -85,B 0,C 180,E1 -3227.526,E2 -3227.526} C_VEL
LIN {X 0,Y 680.478,Z 336.459,A -85,B 0,C 180,E1 -3230.698,E2 -3230.698} C_VEL
LIN {X 0,Y 680.462,Z 336.464,A -85,B 0,C 180,E1 -3233.419,E2 -3233.419} C_VEL
LIN {X 0,Y 680.523,Z 336.461,A -85,B 0,C 180,E1 -3236.378,E2 -3236.378} C_VEL
LIN {X 0,Y 680.457,Z 336.459,A -85,B 0,C 180,E1 -3239.242,E2 -3239.242} C_VEL
LIN {X 0,Y 680.505,Z 336.465,A -85,B 0,C 180,E1 -3242.021,E2 -3242.021} C_VEL
LIN {X 0,Y 680.469,Z 336.462,A -85,B 0,C 180,E1 -3245.058,E2 -3245.058} C_VEL
LIN {X 0,Y 680.462,Z 336.458,A -85,B 0,C 180,E1 -3247.685,E2 -3247.685} C_VEL
LIN {X 0,Y 680.52,Z 336.453,A -85,B 0,C 180,E1 -3250.669,E2 -3250.669} C_VEL
LIN {X 0,Y 680.455,Z 336.464,A -85,B 0,C 180,E1 -3253.512,E2 -3253.512} C_VEL
LIN {X 0,Y 680.508,Z 336.459,A -85,B 0,C 180,E1 -3256.299,E2 -3256.299} C_VEL
LIN {X 0,Y 680.464,Z 336.455,A -85,B 0,C 180,E1 -3259.307,E2 -3259.307} C_VEL
LIN {X 0,Y 680.461,Z 336.465,A -85,B 0,C 180,E1 -3261.915,E2 -3261.915} C_VEL
LIN {X 0,Y 680.526,Z 336.461,A -85,B 0,C 180,E1 -3264.848,E2 -3264.848} C_VEL
LIN {X 0,Y 680.456,Z 336.461,A -85,B 0,C 180,E1 -3267.763,E2 -3267.763} C_VEL
LIN {X 0,Y 680.515,Z 336.466,A -85,B 0,C 180,E1 -3270.569,E2 -3270.569} C_VEL
LIN {X 0,Y 680.466,Z 336.464,A -85,B 0,C 180,E1 -3273.575,E2 -3273.575} C_VEL
LIN {X 0,Y 680.466,Z 336.467,A -85,B 0,C 180,E1 -3276.224,E2 -3276.224} C_VEL
LIN {X 0,Y 680.504,Z 336.463,A -85,B 0,C 180,E1 -3279.293,E2 -3279.293} C_VEL
LIN {X 0,Y 680.456,Z 336.465,A -85,B 0,C 180,E1 -3282.072,E2 -3282.072} C_VEL
LIN {X 0,Y 680.527,Z 336.463,A -85,B 0,C 180,E1 -3284.97,E2 -3284.97} C_VEL
LIN {X 0,Y 680.458,Z 336.468,A -85,B 0,C 180,E1 -3287.928,E2 -3287.928} C_VEL
LIN {X 0,Y 680.49,Z 336.536,A -85,B 0,C 180,E1 -3289.651,E2 -3289.651} C_VEL
LIN {X 0,Y 689.626,Z 360.874,A -85,B 0,C 180,E1 -3292.143,E2 -3292.143} C_VEL
LIN {X 0,Y 689.264,Z 377.17,A -85,B 0,C 180,E1 -3293.327,E2 -3293.327} C_VEL
LIN {X 0,Y 693.662,Z 395.744,A -85,B 0,C 180,E1 -3293.828,E2 -3293.828} C_VEL
LIN {X 0,Y 691.445,Z 657.884,A -85,B 0,C 180,E1 -3296.937,E2 -3296.937} C_VEL
LIN {X 0,Y 690.51,Z 767.576,A -85,B 0,C 180,E1 -3298.238,E2 -3298.238} C_VEL
LIN {X 0,Y 689.952,Z 793.018,A -85,B 0,C 180,E1 -3298.689,E2 -3298.689} C_VEL
LIN {X 0,Y 689.325,Z 814.667,A -85,B 0,C 180,E1 -3299.209,E2 -3299.209} C_VEL
LIN {X 0,Y 688.609,Z 838.554,A -85,B 0,C 180,E1 -3299.937,E2 -3299.937} C_VEL
LIN {X 0,Y 687.794,Z 859.592,A -85,B 0,C 180,E1 -3300.723,E2 -3300.723} C_VEL
LIN {X 0,Y 686.919,Z 881.255,A -85,B 0,C 180,E1 -3301.671,E2 -3301.671} C_VEL
LIN {X 0,Y 685.951,Z 903.052,A -85,B 0,C 180,E1 -3302.803,E2 -3302.803} C_VEL
LIN {X 0,Y 685.057,Z 922.955,A -85,B 0,C 180,E1 -3303.988,E2 -3303.988} C_VEL
LIN {X 0,Y 684.091,Z 943.292,A -85,B 0,C 180,E1 -3305.387,E2 -3305.387} C_VEL
LIN {X 0,Y 683.28,Z 961.609,A -85,B 0,C 180,E1 -3306.818,E2 -3306.818} C_VEL
LIN {X 0,Y 682.482,Z 979.534,A -85,B 0,C 180,E1 -3308.424,E2 -3308.424} C_VEL
LIN {X 0,Y 681.841,Z 995.625,A -85,B 0,C 180,E1 -3310.052,E2 -3310.052} C_VEL
LIN {X 0,Y 681.258,Z 1011.229,A -85,B 0,C 180,E1 -3311.871,E2 -3311.871} C_VEL
LIN {X 0,Y 680.802,Z 1025.061,A -85,B 0,C 180,E1 -3313.709,E2 -3313.709} C_VEL
LIN {X 0,Y 680.459,Z 1037.321,A -85,B 0,C 180,E1 -3315.621,E2 -3315.621} C_VEL
LIN {X 0,Y 680.233,Z 1047.861,A -85,B 0,C 180,E1 -3317.521,E2 -3317.521} C_VEL
LIN {X 0,Y 680.077,Z 1056.896,A -85,B 0,C 180,E1 -3319.496,E2 -3319.496} C_VEL
LIN {X 0,Y 679.969,Z 1063.726,A -85,B 0,C 180,E1 -3321.288,E2 -3321.288} C_VEL
LIN {X 0,Y 679.919,Z 1070.07,A -85,B 0,C 180,E1 -3323.413,E2 -3323.413} C_VEL
LIN {X 0,Y 679.921,Z 1073.974,A -85,B 0,C 180,E1 -3325.192,E2 -3325.192} C_VEL
LIN {X 0,Y 679.908,Z 1077.017,A -85,B 0,C 180,E1 -3327.218,E2 -3327.218} C_VEL
LIN {X 0,Y 679.899,Z 1078.306,A -85,B 0,C 180,E1 -3329.242,E2 -3329.242} C_VEL
LIN {X 0,Y 679.914,Z 1078.238,A -85,B 0,C 180,E1 -3331.011,E2 -3331.011} C_VEL
LIN {X 0,Y 679.916,Z 1076.461,A -85,B 0,C 180,E1 -3333.204,E2 -3333.204} C_VEL
LIN {X 0,Y 679.923,Z 1073.496,A -85,B 0,C 180,E1 -3335.062,E2 -3335.062} C_VEL
LIN {X 0,Y 679.954,Z 1068.507,A -85,B 0,C 180,E1 -3337.18,E2 -3337.18} C_VEL
LIN {X 0,Y 679.992,Z 1062.513,A -85,B 0,C 180,E1 -3339.052,E2 -3339.052} C_VEL
LIN {X 0,Y 680.097,Z 1055.12,A -85,B 0,C 180,E1 -3340.933,E2 -3340.933} C_VEL
LIN {X 0,Y 680.283,Z 1045.255,A -85,B 0,C 180,E1 -3342.969,E2 -3342.969} C_VEL
LIN {X 0,Y 680.52,Z 1035.245,A -85,B 0,C 180,E1 -3344.726,E2 -3344.726} C_VEL
LIN {X 0,Y 680.898,Z 1021.894,A -85,B 0,C 180,E1 -3346.728,E2 -3346.728} C_VEL
LIN {X 0,Y 681.318,Z 1009.107,A -85,B 0,C 180,E1 -3348.393,E2 -3348.393} C_VEL
LIN {X 0,Y 681.951,Z 992.791,A -85,B 0,C 180,E1 -3350.245,E2 -3350.245} C_VEL
LIN {X 0,Y 682.561,Z 977.636,A -85,B 0,C 180,E1 -3351.758,E2 -3351.758} C_VEL
LIN {X 0,Y 683.397,Z 958.847,A -85,B 0,C 180,E1 -3353.405,E2 -3353.405} C_VEL
LIN {X 0,Y 684.206,Z 940.792,A -85,B 0,C 180,E1 -3354.798,E2 -3354.798} C_VEL
LIN {X 0,Y 685.184,Z 919.997,A -85,B 0,C 180,E1 -3356.196,E2 -3356.196} C_VEL
LIN {X 0,Y 686.049,Z 900.695,A -85,B 0,C 180,E1 -3357.329,E2 -3357.329} C_VEL
LIN {X 0,Y 687.089,Z 877.282,A -85,B 0,C 180,E1 -3358.511,E2 -3358.511} C_VEL
LIN {X 0,Y 687.891,Z 857.092,A -85,B 0,C 180,E1 -3359.378,E2 -3359.378} C_VEL
LIN {X 0,Y 688.774,Z 832.985,A -85,B 0,C 180,E1 -3360.248,E2 -3360.248} C_VEL
LIN {X 0,Y 689.455,Z 811.007,A -85,B 0,C 180,E1 -3360.886,E2 -3360.886} C_VEL
LIN {X 0,Y 690.143,Z 786.732,A -85,B 0,C 180,E1 -3361.441,E2 -3361.441} C_VEL
LIN {X 0,Y 690.547,Z 763.43,A -85,B 0,C 180,E1 -3361.819,E2 -3361.819} C_VEL
LIN {X 0,Y 692.558,Z 519.957,A -85,B 0,C 180,E1 -3364.69,E2 -3364.69} C_VEL
LIN {X 0,Y 693.501,Z 394.27,A -85,B 0,C 180,E1 -3366.2,E2 -3366.2} C_VEL
LIN {X 0,Y 689.198,Z 376.448,A -85,B 0,C 180,E1 -3366.707,E2 -3366.707} C_VEL
LIN {X 0,Y 689.442,Z 360.316,A -85,B 0,C 180,E1 -3367.911,E2 -3367.911} C_VEL
LIN {X 0,Y 682.414,Z 342.087,A -85,B 0,C 180,E1 -3369.779,E2 -3369.779} C_VEL
LIN {X 0,Y 680.484,Z 336.477,A -85,B 0,C 180,E1 -3370.363,E2 -3370.363} C_VEL
LIN {X 0,Y 680.477,Z 336.471,A -85,B 0,C 180,E1 -3373.457,E2 -3373.457} C_VEL
LIN {X 0,Y 680.457,Z 336.467,A -85,B 0,C 180,E1 -3376.086,E2 -3376.086} C_VEL
LIN {X 0,Y 680.531,Z 336.466,A -85,B 0,C 180,E1 -3379.057,E2 -3379.057} C_VEL
LIN {X 0,Y 680.456,Z 336.464,A -85,B 0,C 180,E1 -3381.964,E2 -3381.964} C_VEL
LIN {X 0,Y 680.505,Z 336.462,A -85,B 0,C 180,E1 -3384.781,E2 -3384.781} C_VEL
LIN {X 0,Y 680.464,Z 336.464,A -85,B 0,C 180,E1 -3387.864,E2 -3387.864} C_VEL
LIN {X 0,Y 680.466,Z 336.462,A -85,B 0,C 180,E1 -3390.511,E2 -3390.511} C_VEL
LIN {X 0,Y 680.505,Z 336.463,A -85,B 0,C 180,E1 -3393.563,E2 -3393.563} C_VEL
LIN {X 0,Y 680.455,Z 336.457,A -85,B 0,C 180,E1 -3396.349,E2 -3396.349} C_VEL
LIN {X 0,Y 680.524,Z 336.46,A -85,B 0,C 180,E1 -3399.172,E2 -3399.172} C_VEL
LIN {X 0,Y 680.464,Z 336.464,A -85,B 0,C 180,E1 -3402.115,E2 -3402.115} C_VEL
LIN {X 0,Y 680.467,Z 336.46,A -85,B 0,C 180,E1 -3404.75,E2 -3404.75} C_VEL
LIN {X 0,Y 680.508,Z 336.467,A -85,B 0,C 180,E1 -3407.785,E2 -3407.785} C_VEL
LIN {X 0,Y 680.457,Z 336.454,A -85,B 0,C 180,E1 -3410.613,E2 -3410.613} C_VEL
LIN {X 0,Y 680.531,Z 336.461,A -85,B 0,C 180,E1 -3413.504,E2 -3413.504} C_VEL
LIN {X 0,Y 680.46,Z 336.462,A -85,B 0,C 180,E1 -3416.462,E2 -3416.462} C_VEL
LIN {X 0,Y 680.482,Z 336.461,A -85,B 0,C 180,E1 -3419.158,E2 -3419.158} C_VEL
LIN {X 0,Y 680.477,Z 336.466,A -85,B 0,C 180,E1 -3422.309,E2 -3422.309} C_VEL
LIN {X 0,Y 680.461,Z 336.459,A -85,B 0,C 180,E1 -3424.974,E2 -3424.974} C_VEL
LIN {X 0,Y 680.525,Z 336.463,A -85,B 0,C 180,E1 -3427.986,E2 -3427.986} C_VEL
LIN {X 0,Y 680.457,Z 336.454,A -85,B 0,C 180,E1 -3430.841,E2 -3430.841} C_VEL
LIN {X 0,Y 680.516,Z 336.459,A -85,B 0,C 180,E1 -3433.684,E2 -3433.684} C_VEL
LIN {X 0,Y 680.47,Z 336.462,A -85,B 0,C 180,E1 -3436.654,E2 -3436.654} C_VEL
LIN {X 0,Y 680.473,Z 336.461,A -85,B 0,C 180,E1 -3439.377,E2 -3439.377} C_VEL
LIN {X 0,Y 680.501,Z 336.467,A -85,B 0,C 180,E1 -3442.46,E2 -3442.46} C_VEL
LIN {X 0,Y 680.458,Z 336.455,A -85,B 0,C 180,E1 -3445.223,E2 -3445.223} C_VEL
LIN {X 0,Y 680.532,Z 336.463,A -85,B 0,C 180,E1 -3448.168,E2 -3448.168} C_VEL
LIN {X 0,Y 680.52,Z 336.461,A -85,B 0,C 180,E1 -3450.461,E2 -3450.461} C_VEL
LIN {X 0,Y 679.466,Z 336.601,A -85,B 0,C 180,E1 -3451.109,E2 -3451.109} C_VEL
LIN {X 0,Y 673.041,Z 337.385,A -85,B 0,C 180,E1 -3452.927,E2 -3452.927} C_VEL
LIN {X 0,Y 672.523,Z 337.446,A -85,B 0,C 180,E1 -3453.399,E2 -3453.399} C_VEL
LIN {X 0,Y 672.587,Z 337.449,A -85,B 0,C 180,E1 -3456.382,E2 -3456.382} C_VEL
LIN {X 0,Y 672.523,Z 337.451,A -85,B 0,C 180,E1 -3459.299,E2 -3459.299} C_VEL
LIN {X 0,Y 672.573,Z 337.452,A -85,B 0,C 180,E1 -3462.111,E2 -3462.111} C_VEL
LIN {X 0,Y 672.529,Z 337.444,A -85,B 0,C 180,E1 -3465.193,E2 -3465.193} C_VEL
LIN {X 0,Y 672.538,Z 337.449,A -85,B 0,C 180,E1 -3467.893,E2 -3467.893} C_VEL
LIN {X 0,Y 672.553,Z 337.459,A -85,B 0,C 180,E1 -3471.037,E2 -3471.037} C_VEL
LIN {X 0,Y 672.551,Z 337.617,A -85,B 0,C 180,E1 -3473.38,E2 -3473.38} C_VEL
LIN {X 0,Y 676.581,Z 348.492,A -85,B 0,C 180,E1 -3474.573,E2 -3474.573} C_VEL
LIN {X 0,Y 686.819,Z 366.483,A -85,B 0,C 180,E1 -3475.46,E2 -3475.46} C_VEL
LIN {X 0,Y 687.145,Z 369.523,A -85,B 0,C 180,E1 -3475.519,E2 -3475.519} C_VEL
LIN {X 0,Y 684.937,Z 605.975,A -85,B 0,C 180,E1 -3478.357,E2 -3478.357} C_VEL
LIN {X 0,Y 683.701,Z 737.454,A -85,B 0,C 180,E1 -3479.927,E2 -3479.927} C_VEL
LIN {X 0,Y 683.098,Z 762.982,A -85,B 0,C 180,E1 -3480.383,E2 -3480.383} C_VEL
LIN {X 0,Y 682.418,Z 784.428,A -85,B 0,C 180,E1 -3480.901,E2 -3480.901} C_VEL
LIN {X 0,Y 681.594,Z 808.728,A -85,B 0,C 180,E1 -3481.647,E2 -3481.647} C_VEL
LIN {X 0,Y 680.746,Z 828.609,A -85,B 0,C 180,E1 -3482.393,E2 -3482.393} C_VEL
LIN {X 0,Y 679.837,Z 849.314,A -85,B 0,C 180,E1 -3483.3,E2 -3483.3} C_VEL
LIN {X 0,Y 678.703,Z 872.036,A -85,B 0,C 180,E1 -3484.474,E2 -3484.474} C_VEL
LIN {X 0,Y 677.739,Z 891.66,A -85,B 0,C 180,E1 -3485.647,E2 -3485.647} C_VEL
LIN {X 0,Y 676.632,Z 912.524,A -85,B 0,C 180,E1 -3487.084,E2 -3487.084} C_VEL
LIN {X 0,Y 675.764,Z 930.2,A -85,B 0,C 180,E1 -3488.472,E2 -3488.472} C_VEL
LIN {X 0,Y 674.826,Z 949.063,A -85,B 0,C 180,E1 -3490.165,E2 -3490.165} C_VEL
LIN {X 0,Y 674.128,Z 964.72,A -85,B 0,C 180,E1 -3491.762,E2 -3491.762} C_VEL
LIN {X 0,Y 673.443,Z 980.568,A -85,B 0,C 180,E1 -3493.614,E2 -3493.614} C_VEL
LIN {X 0,Y 672.97,Z 993.715,A -85,B 0,C 180,E1 -3495.37,E2 -3495.37} C_VEL
LIN {X 0,Y 672.58,Z 1006.12,A -85,B 0,C 180,E1 -3497.29,E2 -3497.29} C_VEL
LIN {X 0,Y 672.312,Z 1015.81,A -85,B 0,C 180,E1 -3499.026,E2 -3499.026} C_VEL
LIN {X 0,Y 672.106,Z 1025.606,A -85,B 0,C 180,E1 -3501.099,E2 -3501.099} C_VEL
LIN {X 0,Y 672.002,Z 1032.768,A -85,B 0,C 180,E1 -3502.957,E2 -3502.957} C_VEL
LIN {X 0,Y 671.953,Z 1039.052,A -85,B 0,C 180,E1 -3504.963,E2 -3504.963} C_VEL
LIN {X 0,Y 671.917,Z 1043.668,A -85,B 0,C 180,E1 -3507.014,E2 -3507.014} C_VEL
LIN {X 0,Y 671.912,Z 1046.577,A -85,B 0,C 180,E1 -3508.892,E2 -3508.892} C_VEL
LIN {X 0,Y 671.911,Z 1048.239,A -85,B 0,C 180,E1 -3511.023,E2 -3511.023} C_VEL
LIN {X 0,Y 671.901,Z 1048.306,A -85,B 0,C 180,E1 -3512.815,E2 -3512.815} C_VEL
LIN {X 0,Y 671.901,Z 1047.011,A -85,B 0,C 180,E1 -3514.866,E2 -3514.866} C_VEL
LIN {X 0,Y 671.913,Z 1044.111,A -85,B 0,C 180,E1 -3516.837,E2 -3516.837} C_VEL
LIN {X 0,Y 671.93,Z 1040.23,A -85,B 0,C 180,E1 -3518.644,E2 -3518.644} C_VEL
LIN {X 0,Y 671.979,Z 1033.919,A -85,B 0,C 180,E1 -3520.806,E2 -3520.806} C_VEL
LIN {X 0,Y 672.093,Z 1027.074,A -85,B 0,C 180,E1 -3522.632,E2 -3522.632} C_VEL
LIN {X 0,Y 672.28,Z 1018.007,A -85,B 0,C 180,E1 -3524.646,E2 -3524.646} C_VEL
LIN {X 0,Y 672.542,Z 1007.386,A -85,B 0,C 180,E1 -3526.586,E2 -3526.586} C_VEL
LIN {X 0,Y 672.926,Z 995.003,A -85,B 0,C 180,E1 -3528.541,E2 -3528.541} C_VEL
LIN {X 0,Y 673.43,Z 980.998,A -85,B 0,C 180,E1 -3530.421,E2 -3530.421} C_VEL
LIN {X 0,Y 674.098,Z 965.519,A -85,B 0,C 180,E1 -3532.243,E2 -3532.243} C_VEL
LIN {X 0,Y 674.815,Z 949.282,A -85,B 0,C 180,E1 -3533.903,E2 -3533.903} C_VEL
LIN {X 0,Y 675.726,Z 930.994,A -85,B 0,C 180,E1 -3535.553,E2 -3535.553} C_VEL
LIN {X 0,Y 676.583,Z 913.495,A -85,B 0,C 180,E1 -3536.934,E2 -3536.934} C_VEL
LIN {X 0,Y 677.683,Z 892.893,A -85,B 0,C 180,E1 -3538.366,E2 -3538.366} C_VEL
LIN {X 0,Y 678.634,Z 873.594,A -85,B 0,C 180,E1 -3539.528,E2 -3539.528} C_VEL
LIN {X 0,Y 679.741,Z 851.422,A -85,B 0,C 180,E1 -3540.693,E2 -3540.693} C_VEL
LIN {X 0,Y 680.676,Z 830.276,A -85,B 0,C 180,E1 -3541.629,E2 -3541.629} C_VEL
LIN {X 0,Y 681.516,Z 810.536,A -85,B 0,C 180,E1 -3542.379,E2 -3542.379} C_VEL
LIN {X 0,Y 682.396,Z 785.089,A -85,B 0,C 180,E1 -3543.171,E2 -3543.171} C_VEL
LIN {X 0,Y 683.074,Z 763.638,A -85,B 0,C 180,E1 -3543.693,E2 -3543.693} C_VEL
LIN {X 0,Y 683.695,Z 738.242,A -85,B 0,C 180,E1 -3544.152,E2 -3544.152} C_VEL
LIN {X 0,Y 684.491,Z 656.49,A -85,B 0,C 180,E1 -3545.136,E2 -3545.136} C_VEL
LIN {X 0,Y 686.779,Z 406.71,A -85,B 0,C 180,E1 -3548.12,E2 -3548.12} C_VEL
LIN {X 0,Y 686.991,Z 367.172,A -85,B 0,C 180,E1 -3548.61,E2 -3548.61} C_VEL
LIN {X 0,Y 685.188,Z 363.29,A -85,B 0,C 180,E1 -3548.773,E2 -3548.773} C_VEL
LIN {X 0,Y 676.327,Z 347.874,A -85,B 0,C 180,E1 -3549.563,E2 -3549.563} C_VEL
LIN {X 0,Y 672.529,Z 337.459,A -85,B 0,C 180,E1 -3550.745,E2 -3550.745} C_VEL
LIN {X 0,Y 672.582,Z 337.45,A -85,B 0,C 180,E1 -3553.738,E2 -3553.738} C_VEL
LIN {X 0,Y 672.521,Z 337.451,A -85,B 0,C 180,E1 -3556.638,E2 -3556.638} C_VEL
LIN {X 0,Y 672.589,Z 337.433,A -85,B 0,C 180,E1 -3559.596,E2 -3559.596} C_VEL
LIN {X 0,Y 672.522,Z 337.452,A -85,B 0,C 180,E1 -3562.555,E2 -3562.555} C_VEL
LIN {X 0,Y 672.565,Z 337.438,A -85,B 0,C 180,E1 -3565.395,E2 -3565.395} C_VEL
LIN {X 0,Y 672.531,Z 337.446,A -85,B 0,C 180,E1 -3568.443,E2 -3568.443} C_VEL
LIN {X 0,Y 672.53,Z 337.454,A -85,B 0,C 180,E1 -3571.128,E2 -3571.128} C_VEL
LIN {X 0,Y 672.568,Z 337.445,A -85,B 0,C 180,E1 -3574.177,E2 -3574.177} C_VEL
LIN {X 0,Y 672.52,Z 337.454,A -85,B 0,C 180,E1 -3576.982,E2 -3576.982} C_VEL
LIN {X 0,Y 672.592,Z 337.453,A -85,B 0,C 180,E1 -3579.915,E2 -3579.915} C_VEL
LIN {X 0,Y 672.52,Z 337.449,A -85,B 0,C 180,E1 -3582.879,E2 -3582.879} C_VEL
LIN {X 0,Y 672.551,Z 337.453,A -85,B 0,C 180,E1 -3585.624,E2 -3585.624} C_VEL
LIN {X 0,Y 672.532,Z 337.45,A -85,B 0,C 180,E1 -3588.769,E2 -3588.769} C_VEL
LIN {X 0,Y 672.528,Z 337.451,A -85,B 0,C 180,E1 -3591.45,E2 -3591.45} C_VEL
LIN {X 0,Y 672.576,Z 337.446,A -85,B 0,C 180,E1 -3594.455,E2 -3594.455} C_VEL
LIN {X 0,Y 672.517,Z 337.453,A -85,B 0,C 180,E1 -3597.273,E2 -3597.273} C_VEL
LIN {X 0,Y 672.59,Z 337.453,A -85,B 0,C 180,E1 -3600.17,E2 -3600.17} C_VEL
LIN {X 0,Y 672.522,Z 337.445,A -85,B 0,C 180,E1 -3603.153,E2 -3603.153} C_VEL
LIN {X 0,Y 672.542,Z 337.456,A -85,B 0,C 180,E1 -3605.888,E2 -3605.888} C_VEL
LIN {X 0,Y 672.534,Z 337.451,A -85,B 0,C 180,E1 -3609.067,E2 -3609.067} C_VEL
LIN {X 0,Y 672.522,Z 337.446,A -85,B 0,C 180,E1 -3611.753,E2 -3611.753} C_VEL
LIN {X 0,Y 672.586,Z 337.441,A -85,B 0,C 180,E1 -3614.727,E2 -3614.727} C_VEL
LIN {X 0,Y 672.517,Z 337.453,A -85,B 0,C 180,E1 -3617.63,E2 -3617.63} C_VEL
LIN {X 0,Y 672.585,Z 337.45,A -85,B 0,C 180,E1 -3620.539,E2 -3620.539} C_VEL
LIN {X 0,Y 672.521,Z 337.445,A -85,B 0,C 180,E1 -3623.482,E2 -3623.482} C_VEL
LIN {X 0,Y 672.539,Z 337.455,A -85,B 0,C 180,E1 -3626.204,E2 -3626.204} C_VEL
LIN {X 0,Y 672.535,Z 337.45,A -85,B 0,C 180,E1 -3629.398,E2 -3629.398} C_VEL
LIN {X 0,Y 672.521,Z 337.455,A -85,B 0,C 180,E1 -3632.063,E2 -3632.063} C_VEL
LIN {X 0,Y 672.584,Z 337.452,A -85,B 0,C 180,E1 -3635.019,E2 -3635.019} C_VEL
LIN {X 0,Y 672.517,Z 337.453,A -85,B 0,C 180,E1 -3637.883,E2 -3637.883} C_VEL
LIN {X 0,Y 672.567,Z 337.455,A -85,B 0,C 180,E1 -3640.694,E2 -3640.694} C_VEL
LIN {X 0,Y 672.526,Z 337.453,A -85,B 0,C 180,E1 -3643.737,E2 -3643.737} C_VEL
LIN {X 0,Y 672.526,Z 337.458,A -85,B 0,C 180,E1 -3646.391,E2 -3646.391} C_VEL
LIN {X 0,Y 672.592,Z 337.467,A -85,B 0,C 180,E1 -3649.174,E2 -3649.174} C_VEL
LIN {X 0,Y 682.601,Z 364.163,A -85,B 0,C 180,E1 -3651.955,E2 -3651.955} C_VEL
LIN {X 0,Y 682.307,Z 376.941,A -85,B 0,C 180,E1 -3652.891,E2 -3652.891} C_VEL
LIN {X 0,Y 687.167,Z 397.582,A -85,B 0,C 180,E1 -3653.458,E2 -3653.458} C_VEL
LIN {X 0,Y 684.716,Z 660.338,A -85,B 0,C 180,E1 -3656.6,E2 -3656.6} C_VEL
LIN {X 0,Y 683.699,Z 767.71,A -85,B 0,C 180,E1 -3657.886,E2 -3657.886} C_VEL
LIN {X 0,Y 683.091,Z 793.146,A -85,B 0,C 180,E1 -3658.342,E2 -3658.342} C_VEL
LIN {X 0,Y 682.412,Z 814.556,A -85,B 0,C 180,E1 -3658.86,E2 -3658.86} C_VEL
LIN {X 0,Y 681.585,Z 838.968,A -85,B 0,C 180,E1 -3659.61,E2 -3659.61} C_VEL
LIN {X 0,Y 680.717,Z 859.347,A -85,B 0,C 180,E1 -3660.378,E2 -3660.378} C_VEL
LIN {X 0,Y 679.794,Z 880.266,A -85,B 0,C 180,E1 -3661.299,E2 -3661.299} C_VEL
LIN {X 0,Y 678.692,Z 902.317,A -85,B 0,C 180,E1 -3662.445,E2 -3662.445} C_VEL
LIN {X 0,Y 677.757,Z 921.216,A -85,B 0,C 180,E1 -3663.574,E2 -3663.574} C_VEL
LIN {X 0,Y 676.663,Z 942.008,A -85,B 0,C 180,E1 -3665,E2 -3665} C_VEL
LIN {X 0,Y 675.802,Z 959.4,A -85,B 0,C 180,E1 -3666.362,E2 -3666.362} C_VEL
LIN {X 0,Y 674.844,Z 978.606,A -85,B 0,C 180,E1 -3668.076,E2 -3668.076} C_VEL
LIN {X 0,Y 674.17,Z 993.722,A -85,B 0,C 180,E1 -3669.611,E2 -3669.611} C_VEL
LIN {X 0,Y 673.468,Z 1009.816,A -85,B 0,C 180,E1 -3671.475,E2 -3671.475} C_VEL
LIN {X 0,Y 673.008,Z 1022.525,A -85,B 0,C 180,E1 -3673.159,E2 -3673.159} C_VEL
LIN {X 0,Y 672.584,Z 1035.764,A -85,B 0,C 180,E1 -3675.185,E2 -3675.185} C_VEL
LIN {X 0,Y 672.325,Z 1045.586,A -85,B 0,C 180,E1 -3676.939,E2 -3676.939} C_VEL
LIN {X 0,Y 672.117,Z 1055.476,A -85,B 0,C 180,E1 -3679.023,E2 -3679.023} C_VEL
LIN {X 0,Y 672.012,Z 1062.514,A -85,B 0,C 180,E1 -3680.839,E2 -3680.839} C_VEL
LIN {X 0,Y 671.958,Z 1068.761,A -85,B 0,C 180,E1 -3682.82,E2 -3682.82} C_VEL
LIN {X 0,Y 671.924,Z 1073.497,A -85,B 0,C 180,E1 -3684.877,E2 -3684.877} C_VEL
LIN {X 0,Y 671.916,Z 1076.462,A -85,B 0,C 180,E1 -3686.758,E2 -3686.758} C_VEL
LIN {X 0,Y 671.914,Z 1078.238,A -85,B 0,C 180,E1 -3688.977,E2 -3688.977} C_VEL
LIN {X 0,Y 671.899,Z 1078.306,A -85,B 0,C 180,E1 -3690.767,E2 -3690.767} C_VEL
LIN {X 0,Y 671.909,Z 1077.017,A -85,B 0,C 180,E1 -3692.815,E2 -3692.815} C_VEL
LIN {X 0,Y 671.922,Z 1073.974,A -85,B 0,C 180,E1 -3694.866,E2 -3694.866} C_VEL
LIN {X 0,Y 671.923,Z 1070.07,A -85,B 0,C 180,E1 -3696.665,E2 -3696.665} C_VEL
LIN {X 0,Y 671.979,Z 1063.726,A -85,B 0,C 180,E1 -3698.816,E2 -3698.816} C_VEL
LIN {X 0,Y 672.097,Z 1056.896,A -85,B 0,C 180,E1 -3700.631,E2 -3700.631} C_VEL
LIN {X 0,Y 672.282,Z 1047.686,A -85,B 0,C 180,E1 -3702.662,E2 -3702.662} C_VEL
LIN {X 0,Y 672.539,Z 1037.261,A -85,B 0,C 180,E1 -3704.563,E2 -3704.563} C_VEL
LIN {X 0,Y 672.919,Z 1025.063,A -85,B 0,C 180,E1 -3706.488,E2 -3706.488} C_VEL
LIN {X 0,Y 673.423,Z 1011.227,A -85,B 0,C 180,E1 -3708.347,E2 -3708.347} C_VEL
LIN {X 0,Y 674.071,Z 996.17,A -85,B 0,C 180,E1 -3710.129,E2 -3710.129} C_VEL
LIN {X 0,Y 674.76,Z 980.459,A -85,B 0,C 180,E1 -3711.744,E2 -3711.744} C_VEL
LIN {X 0,Y 675.65,Z 962.715,A -85,B 0,C 180,E1 -3713.366,E2 -3713.366} C_VEL
LIN {X 0,Y 676.557,Z 944.067,A -85,B 0,C 180,E1 -3714.846,E2 -3714.846} C_VEL
LIN {X 0,Y 677.598,Z 924.668,A -85,B 0,C 180,E1 -3716.208,E2 -3716.208} C_VEL
LIN {X 0,Y 678.618,Z 903.936,A -85,B 0,C 180,E1 -3717.463,E2 -3717.463} C_VEL
LIN {X 0,Y 679.681,Z 882.64,A -85,B 0,C 180,E1 -3718.59,E2 -3718.59} C_VEL
LIN {X 0,Y 680.68,Z 860.265,A -85,B 0,C 180,E1 -3719.585,E2 -3719.585} C_VEL
LIN {X 0,Y 681.547,Z 839.834,A -85,B 0,C 180,E1 -3720.359,E2 -3720.359} C_VEL
LIN {X 0,Y 682.405,Z 814.776,A -85,B 0,C 180,E1 -3721.134,E2 -3721.134} C_VEL
LIN {X 0,Y 683.086,Z 793.282,A -85,B 0,C 180,E1 -3721.656,E2 -3721.656} C_VEL
LIN {X 0,Y 683.699,Z 767.822,A -85,B 0,C 180,E1 -3722.113,E2 -3722.113} C_VEL
LIN {X 0,Y 684.658,Z 666.935,A -85,B 0,C 180,E1 -3723.322,E2 -3723.322} C_VEL
LIN {X 0,Y 687.132,Z 401.239,A -85,B 0,C 180,E1 -3726.498,E2 -3726.498} C_VEL
LIN {X 0,Y 686.935,Z 395.795,A -85,B 0,C 180,E1 -3726.58,E2 -3726.58} C_VEL
LIN {X 0,Y 682.24,Z 376.221,A -85,B 0,C 180,E1 -3727.144,E2 -3727.144} C_VEL
LIN {X 0,Y 682.47,Z 363.779,A -85,B 0,C 180,E1 -3728.083,E2 -3728.083} C_VEL
LIN {X 0,Y 674.923,Z 343.947,A -85,B 0,C 180,E1 -3730.142,E2 -3730.142} C_VEL
LIN {X 0,Y 672.591,Z 337.458,A -85,B 0,C 180,E1 -3730.852,E2 -3730.852} C_VEL
LIN {X 0,Y 672.521,Z 337.459,A -85,B 0,C 180,E1 -3733.737,E2 -3733.737} C_VEL
LIN {X 0,Y 672.537,Z 337.455,A -85,B 0,C 180,E1 -3736.389,E2 -3736.389} C_VEL
LIN {X 0,Y 672.535,Z 337.451,A -85,B 0,C 180,E1 -3739.592,E2 -3739.592} C_VEL
LIN {X 0,Y 672.521,Z 337.451,A -85,B 0,C 180,E1 -3742.276,E2 -3742.276} C_VEL
LIN {X 0,Y 672.58,Z 337.449,A -85,B 0,C 180,E1 -3745.297,E2 -3745.297} C_VEL
LIN {X 0,Y 672.515,Z 337.451,A -85,B 0,C 180,E1 -3748.142,E2 -3748.142} C_VEL
LIN {X 0,Y 672.574,Z 337.449,A -85,B 0,C 180,E1 -3750.945,E2 -3750.945} C_VEL
LIN {X 0,Y 672.526,Z 337.454,A -85,B 0,C 180,E1 -3753.985,E2 -3753.985} C_VEL
LIN {X 0,Y 672.535,Z 337.443,A -85,B 0,C 180,E1 -3756.704,E2 -3756.704} C_VEL
LIN {X 0,Y 672.538,Z 337.449,A -85,B 0,C 180,E1 -3759.913,E2 -3759.913} C_VEL
LIN {X 0,Y 672.525,Z 337.451,A -85,B 0,C 180,E1 -3762.651,E2 -3762.651} C_VEL
LIN {X 0,Y 672.574,Z 337.446,A -85,B 0,C 180,E1 -3765.713,E2 -3765.713} C_VEL
LIN {X 0,Y 672.518,Z 337.452,A -85,B 0,C 180,E1 -3768.508,E2 -3768.508} C_VEL
LIN {X 0,Y 672.582,Z 337.44,A -85,B 0,C 180,E1 -3771.364,E2 -3771.364} C_VEL
LIN {X 0,Y 672.525,Z 337.449,A -85,B 0,C 180,E1 -3774.369,E2 -3774.369} C_VEL
LIN {X 0,Y 672.541,Z 337.447,A -85,B 0,C 180,E1 -3777.103,E2 -3777.103} C_VEL
LIN {X 0,Y 672.538,Z 337.444,A -85,B 0,C 180,E1 -3780.256,E2 -3780.256} C_VEL
LIN {X 0,Y 672.525,Z 337.451,A -85,B 0,C 180,E1 -3782.983,E2 -3782.983} C_VEL
LIN {X 0,Y 672.583,Z 337.444,A -85,B 0,C 180,E1 -3785.978,E2 -3785.978} C_VEL
LIN {X 0,Y 672.519,Z 337.453,A -85,B 0,C 180,E1 -3788.809,E2 -3788.809} C_VEL
LIN {X 0,Y 672.576,Z 337.439,A -85,B 0,C 180,E1 -3791.665,E2 -3791.665} C_VEL
LIN {X 0,Y 672.529,Z 337.451,A -85,B 0,C 180,E1 -3794.64,E2 -3794.64} C_VEL
LIN {X 0,Y 672.537,Z 337.447,A -85,B 0,C 180,E1 -3797.388,E2 -3797.388} C_VEL
LIN {X 0,Y 672.546,Z 337.446,A -85,B 0,C 180,E1 -3800.54,E2 -3800.54} C_VEL
LIN {X 0,Y 672.527,Z 337.452,A -85,B 0,C 180,E1 -3803.296,E2 -3803.296} C_VEL
LIN {X 0,Y 672.585,Z 337.446,A -85,B 0,C 180,E1 -3806.306,E2 -3806.306} C_VEL
LIN {X 0,Y 672.522,Z 337.445,A -85,B 0,C 180,E1 -3809.187,E2 -3809.187} C_VEL
LIN {X 0,Y 672.585,Z 337.45,A -85,B 0,C 180,E1 -3812.072,E2 -3812.072} C_VEL
LIN {X 0,Y 672.523,Z 337.446,A -85,B 0,C 180,E1 -3813.399,E2 -3813.399} C_VEL
LIN {X 0,Y 671.558,Z 337.57,A -85,B 0,C 180,E1 -3814.055,E2 -3814.055} C_VEL
LIN {X 0,Y 665.187,Z 338.373,A -85,B 0,C 180,E1 -3815.895,E2 -3815.895} C_VEL
LIN {X 0,Y 664.648,Z 338.437,A -85,B 0,C 180,E1 -3816.373,E2 -3816.373} C_VEL
LIN {X 0,Y 664.585,Z 338.44,A -85,B 0,C 180,E1 -3819.302,E2 -3819.302} C_VEL
LIN {X 0,Y 664.638,Z 338.441,A -85,B 0,C 180,E1 -3822.142,E2 -3822.142} C_VEL
LIN {X 0,Y 664.596,Z 338.429,A -85,B 0,C 180,E1 -3825.123,E2 -3825.123} C_VEL
LIN {X 0,Y 664.598,Z 338.439,A -85,B 0,C 180,E1 -3827.879,E2 -3827.879} C_VEL
LIN {X 0,Y 664.611,Z 338.448,A -85,B 0,C 180,E1 -3831.061,E2 -3831.061} C_VEL
LIN {X 0,Y 664.652,Z 338.576,A -85,B 0,C 180,E1 -3832.897,E2 -3832.897} C_VEL
LIN {X 0,Y 668.468,Z 348.792,A -85,B 0,C 180,E1 -3834.039,E2 -3834.039} C_VEL
LIN {X 0,Y 680.723,Z 370.08,A -85,B 0,C 180,E1 -3835.122,E2 -3835.122} C_VEL
LIN {X 0,Y 678.272,Z 606.578,A -85,B 0,C 180,E1 -3837.988,E2 -3837.988} C_VEL
LIN {X 0,Y 676.917,Z 737.51,A -85,B 0,C 180,E1 -3839.567,E2 -3839.567} C_VEL
LIN {X 0,Y 676.265,Z 763.04,A -85,B 0,C 180,E1 -3840.027,E2 -3840.027} C_VEL
LIN {X 0,Y 675.538,Z 784.266,A -85,B 0,C 180,E1 -3840.544,E2 -3840.544} C_VEL
LIN {X 0,Y 674.669,Z 807.51,A -85,B 0,C 180,E1 -3841.254,E2 -3841.254} C_VEL
LIN {X 0,Y 673.656,Z 829.251,A -85,B 0,C 180,E1 -3842.077,E2 -3842.077} C_VEL
LIN {X 0,Y 672.621,Z 850.868,A -85,B 0,C 180,E1 -3843.038,E2 -3843.038} C_VEL
LIN {X 0,Y 671.416,Z 872.5,A -85,B 0,C 180,E1 -3844.177,E2 -3844.177} C_VEL
LIN {X 0,Y 670.363,Z 892.083,A -85,B 0,C 180,E1 -3845.361,E2 -3845.361} C_VEL
LIN {X 0,Y 669.153,Z 912.814,A -85,B 0,C 180,E1 -3846.808,E2 -3846.808} C_VEL
LIN {X 0,Y 668.189,Z 930.522,A -85,B 0,C 180,E1 -3848.216,E2 -3848.216} C_VEL
LIN {X 0,Y 667.206,Z 948.416,A -85,B 0,C 180,E1 -3849.838,E2 -3849.838} C_VEL
LIN {X 0,Y 666.442,Z 963.293,A -85,B 0,C 180,E1 -3851.363,E2 -3851.363} C_VEL
LIN {X 0,Y 665.641,Z 980.076,A -85,B 0,C 180,E1 -3853.327,E2 -3853.327} C_VEL
LIN {X 0,Y 665.148,Z 992.639,A -85,B 0,C 180,E1 -3855.015,E2 -3855.015} C_VEL
LIN {X 0,Y 664.658,Z 1006.176,A -85,B 0,C 180,E1 -3857.119,E2 -3857.119} C_VEL
LIN {X 0,Y 664.357,Z 1015.988,A -85,B 0,C 180,E1 -3858.902,E2 -3858.902} C_VEL
LIN {X 0,Y 664.129,Z 1025.709,A -85,B 0,C 180,E1 -3860.992,E2 -3860.992} C_VEL
LIN {X 0,Y 664.025,Z 1032.677,A -85,B 0,C 180,E1 -3862.82,E2 -3862.82} C_VEL
LIN {X 0,Y 663.955,Z 1038.873,A -85,B 0,C 180,E1 -3864.816,E2 -3864.816} C_VEL
LIN {X 0,Y 663.92,Z 1043.554,A -85,B 0,C 180,E1 -3866.892,E2 -3866.892} C_VEL
LIN {X 0,Y 663.911,Z 1046.385,A -85,B 0,C 180,E1 -3868.706,E2 -3868.706} C_VEL
LIN {X 0,Y 663.912,Z 1048.199,A -85,B 0,C 180,E1 -3870.863,E2 -3870.863} C_VEL
LIN {X 0,Y 663.899,Z 1048.322,A -85,B 0,C 180,E1 -3872.762,E2 -3872.762} C_VEL
LIN {X 0,Y 663.898,Z 1047.134,A -85,B 0,C 180,E1 -3874.752,E2 -3874.752} C_VEL
LIN {X 0,Y 663.913,Z 1044.224,A -85,B 0,C 180,E1 -3876.833,E2 -3876.833} C_VEL
LIN {X 0,Y 663.933,Z 1040.377,A -85,B 0,C 180,E1 -3878.662,E2 -3878.662} C_VEL
LIN {X 0,Y 663.986,Z 1034.441,A -85,B 0,C 180,E1 -3880.762,E2 -3880.762} C_VEL
LIN {X 0,Y 664.109,Z 1027.328,A -85,B 0,C 180,E1 -3882.698,E2 -3882.698} C_VEL
LIN {X 0,Y 664.305,Z 1018.729,A -85,B 0,C 180,E1 -3884.647,E2 -3884.647} C_VEL
LIN {X 0,Y 664.592,Z 1008.272,A -85,B 0,C 180,E1 -3886.61,E2 -3886.61} C_VEL
LIN {X 0,Y 664.959,Z 997.182,A -85,B 0,C 180,E1 -3888.408,E2 -3888.408} C_VEL
LIN {X 0,Y 665.538,Z 982.914,A -85,B 0,C 180,E1 -3890.399,E2 -3890.399} C_VEL
LIN {X 0,Y 666.139,Z 969.457,A -85,B 0,C 180,E1 -3892.04,E2 -3892.04} C_VEL
LIN {X 0,Y 667.005,Z 952.253,A -85,B 0,C 180,E1 -3893.875,E2 -3893.875} C_VEL
LIN {X 0,Y 667.84,Z 936.516,A -85,B 0,C 180,E1 -3895.353,E2 -3895.353} C_VEL
LIN {X 0,Y 668.968,Z 916.216,A -85,B 0,C 180,E1 -3897.025,E2 -3897.025} C_VEL
LIN {X 0,Y 670.033,Z 897.67,A -85,B 0,C 180,E1 -3898.359,E2 -3898.359} C_VEL
LIN {X 0,Y 671.267,Z 875.582,A -85,B 0,C 180,E1 -3899.737,E2 -3899.737} C_VEL
LIN {X 0,Y 672.336,Z 855.537,A -85,B 0,C 180,E1 -3900.82,E2 -3900.82} C_VEL
LIN {X 0,Y 673.539,Z 831.903,A -85,B 0,C 180,E1 -3901.904,E2 -3901.904} C_VEL
LIN {X 0,Y 674.443,Z 812.39,A -85,B 0,C 180,E1 -3902.659,E2 -3902.659} C_VEL
LIN {X 0,Y 675.396,Z 788.595,A -85,B 0,C 180,E1 -3903.43,E2 -3903.43} C_VEL
LIN {X 0,Y 676.156,Z 765.864,A -85,B 0,C 180,E1 -3904.001,E2 -3904.001} C_VEL
LIN {X 0,Y 676.874,Z 741.591,A -85,B 0,C 180,E1 -3904.465,E2 -3904.465} C_VEL
LIN {X 0,Y 677.412,Z 695.138,A -85,B 0,C 180,E1 -3905.047,E2 -3905.047} C_VEL
LIN {X 0,Y 679.97,Z 442.631,A -85,B 0,C 180,E1 -3908.08,E2 -3908.08} C_VEL
LIN {X 0,Y 680.612,Z 369.671,A -85,B 0,C 180,E1 -3908.98,E2 -3908.98} C_VEL
LIN {X 0,Y 668.308,Z 348.44,A -85,B 0,C 180,E1 -3910.068,E2 -3910.068} C_VEL
LIN {X 0,Y 664.639,Z 338.439,A -85,B 0,C 180,E1 -3911.218,E2 -3911.218} C_VEL
LIN {X 0,Y 664.589,Z 338.441,A -85,B 0,C 180,E1 -3914.275,E2 -3914.275} C_VEL
LIN {X 0,Y 664.604,Z 338.442,A -85,B 0,C 180,E1 -3917.036,E2 -3917.036} C_VEL
LIN {X 0,Y 664.597,Z 338.435,A -85,B 0,C 180,E1 -3920.252,E2 -3920.252} C_VEL
LIN {X 0,Y 664.593,Z 338.44,A -85,B 0,C 180,E1 -3923,E2 -3923} C_VEL
LIN {X 0,Y 664.619,Z 338.439,A -85,B 0,C 180,E1 -3926.146,E2 -3926.146} C_VEL
LIN {X 0,Y 664.585,Z 338.437,A -85,B 0,C 180,E1 -3928.932,E2 -3928.932} C_VEL
LIN {X 0,Y 664.653,Z 338.437,A -85,B 0,C 180,E1 -3931.909,E2 -3931.909} C_VEL
LIN {X 0,Y 664.58,Z 338.436,A -85,B 0,C 180,E1 -3934.799,E2 -3934.799} C_VEL
LIN {X 0,Y 664.631,Z 338.441,A -85,B 0,C 180,E1 -3937.628,E2 -3937.628} C_VEL
LIN {X 0,Y 664.592,Z 338.44,A -85,B 0,C 180,E1 -3940.671,E2 -3940.671} C_VEL
LIN {X 0,Y 664.597,Z 338.441,A -85,B 0,C 180,E1 -3943.41,E2 -3943.41} C_VEL
LIN {X 0,Y 664.604,Z 338.437,A -85,B 0,C 180,E1 -3946.603,E2 -3946.603} C_VEL
LIN {X 0,Y 664.584,Z 338.442,A -85,B 0,C 180,E1 -3949.335,E2 -3949.335} C_VEL
LIN {X 0,Y 664.645,Z 338.437,A -85,B 0,C 180,E1 -3952.392,E2 -3952.392} C_VEL
LIN {X 0,Y 664.579,Z 338.438,A -85,B 0,C 180,E1 -3955.253,E2 -3955.253} C_VEL
LIN {X 0,Y 664.647,Z 338.434,A -85,B 0,C 180,E1 -3958.19,E2 -3958.19} C_VEL
LIN {X 0,Y 664.585,Z 338.441,A -85,B 0,C 180,E1 -3961.121,E2 -3961.121} C_VEL
LIN {X 0,Y 664.606,Z 338.437,A -85,B 0,C 180,E1 -3963.882,E2 -3963.882} C_VEL
LIN {X 0,Y 664.596,Z 338.431,A -85,B 0,C 180,E1 -3967,E2 -3967} C_VEL
LIN {X 0,Y 664.584,Z 338.443,A -85,B 0,C 180,E1 -3969.701,E2 -3969.701} C_VEL
LIN {X 0,Y 664.636,Z 338.438,A -85,B 0,C 180,E1 -3972.777,E2 -3972.777} C_VEL
LIN {X 0,Y 664.578,Z 338.434,A -85,B 0,C 180,E1 -3975.624,E2 -3975.624} C_VEL
LIN {X 0,Y 664.651,Z 338.433,A -85,B 0,C 180,E1 -3978.598,E2 -3978.598} C_VEL
LIN {X 0,Y 664.58,Z 338.442,A -85,B 0,C 180,E1 -3981.595,E2 -3981.595} C_VEL
LIN {X 0,Y 664.631,Z 338.438,A -85,B 0,C 180,E1 -3984.439,E2 -3984.439} C_VEL
LIN {X 0,Y 664.587,Z 338.437,A -85,B 0,C 180,E1 -3987.509,E2 -3987.509} C_VEL
LIN {X 0,Y 664.591,Z 338.443,A -85,B 0,C 180,E1 -3990.166,E2 -3990.166} C_VEL
LIN {X 0,Y 664.613,Z 338.441,A -85,B 0,C 180,E1 -3993.308,E2 -3993.308} C_VEL
LIN {X 0,Y 664.58,Z 338.444,A -85,B 0,C 180,E1 -3996.035,E2 -3996.035} C_VEL
LIN {X 0,Y 664.653,Z 338.44,A -85,B 0,C 180,E1 -3998.964,E2 -3998.964} C_VEL
LIN {X 0,Y 664.579,Z 338.443,A -85,B 0,C 180,E1 -4001.915,E2 -4001.915} C_VEL
LIN {X 0,Y 664.627,Z 338.442,A -85,B 0,C 180,E1 -4004.757,E2 -4004.757} C_VEL
LIN {X 0,Y 664.585,Z 338.443,A -85,B 0,C 180,E1 -4007.854,E2 -4007.854} C_VEL
LIN {X 0,Y 664.621,Z 338.542,A -85,B 0,C 180,E1 -4008.683,E2 -4008.683} C_VEL
LIN {X 0,Y 673.506,Z 362.08,A -85,B 0,C 180,E1 -4011.208,E2 -4011.208} C_VEL
